C05453=1086.280,20.967,-58.503,174.648,18.923,153.065
C05454=1086.286,21.217,-58.517,174.650,18.926,153.065
C05455=1086.291,21.466,-58.532,174.652,18.928,153.065
C05456=1086.298,21.715,-58.547,174.653,18.929,153.065
C05457=1086.303,21.965,-58.562,174.654,18.931,153.065
C05458=1086.309,22.215,-58.576,174.656,18.933,153.065
C05459=1086.315,22.464,-58.591,174.658,18.935,153.065
C05460=1086.320,22.714,-58.606,174.659,18.937,153.065
C05461=1086.326,22.963,-58.621,174.661,18.939,153.065
C05462=1086.332,23.213,-58.635,174.663,18.941,153.066
C05463=1086.337,23.462,-58.650,174.664,18.942,153.066
C05464=1086.344,23.712,-58.665,174.666,18.944,153.066
C05465=1086.349,23.961,-58.680,174.667,18.946,153.066
C05466=1086.354,24.210,-58.695,174.669,18.948,153.066
C05467=1086.361,24.460,-58.710,174.671,18.951,153.066
C05468=1086.366,24.709,-58.724,174.672,18.952,153.066
C05469=1086.372,24.959,-58.739,174.674,18.954,153.066
C05470=1086.378,25.208,-58.754,174.676,18.956,153.066
C05471=1086.384,25.458,-58.769,174.677,18.958,153.066
C05472=1086.389,25.707,-58.784,174.680,18.960,153.066
C05473=1086.395,25.957,-58.799,174.681,18.962,153.066
C05474=1086.401,26.206,-58.813,174.682,18.963,153.067
C05475=1086.407,26.456,-58.829,174.684,18.966,153.067
C05476=1086.412,26.705,-58.843,174.686,18.967,153.067
C05477=1086.419,26.955,-58.858,174.687,18.969,153.067
C05478=1086.424,27.205,-58.873,174.689,18.971,153.067
C05479=1086.430,27.454,-58.888,174.691,18.973,153.067
C05480=1086.436,27.704,-58.903,174.692,18.975,153.067
C05481=1086.442,27.953,-58.918,174.694,18.977,153.067
C05482=1086.448,28.203,-58.933,174.695,18.979,153.067
C05483=1086.453,28.452,-58.948,174.697,18.980,153.067
C05484=1086.459,28.702,-58.963,174.699,18.983,153.067
C05485=1086.464,28.951,-58.978,174.700,18.984,153.067
C05486=1086.471,29.200,-58.993,174.702,18.986,153.068
C05487=1086.476,29.450,-59.008,174.704,18.988,153.068
C05488=1086.482,29.699,-59.023,174.705,18.990,153.068
C05489=1086.487,29.949,-59.038,174.706,18.992,153.068
C05490=1086.494,30.198,-59.053,174.709,18.994,153.068
C05491=1086.499,30.448,-59.069,174.710,18.996,153.068
C05492=1086.505,30.697,-59.084,174.711,18.997,153.068
C05493=1086.512,30.975,-59.101,174.713,19.000,153.068
C05494=1086.518,31.253,-59.117,174.716,19.002,153.068
C05495=1086.524,31.531,-59.134,174.717,19.004,153.068
C05496=1086.530,31.809,-59.152,174.719,19.006,153.068
C05497=1086.536,32.058,-59.167,174.720,19.008,153.069
C05498=1086.542,32.308,-59.182,174.723,19.010,153.069
C05499=1086.548,32.557,-59.197,174.724,19.012,153.069
C05500=1086.554,32.807,-59.212,174.725,19.014,153.069
C05501=1086.559,33.056,-59.227,174.728,19.016,153.069
C05502=1086.565,33.306,-59.242,174.729,19.017,153.069
C05503=1086.571,33.555,-59.257,174.731,19.020,153.069
C05504=1086.576,33.805,-59.272,174.732,19.021,153.069
C05505=1086.582,34.055,-59.288,174.734,19.023,153.069
C05506=1086.588,34.303,-59.303,174.736,19.025,153.069
C05507=1086.594,34.553,-59.319,174.737,19.027,153.069
C05508=1086.600,34.802,-59.333,174.739,19.029,153.069
C05509=1086.605,35.052,-59.349,174.741,19.031,153.069
C05510=1086.612,35.302,-59.364,174.742,19.033,153.070
C05511=1086.617,35.551,-59.380,174.745,19.035,153.070
C05512=1086.623,35.801,-59.395,174.746,19.037,153.070
C05513=1086.629,36.050,-59.410,174.747,19.038,153.070
C05514=1086.634,36.299,-59.425,174.750,19.040,153.070
C05515=1086.640,36.549,-59.440,174.751,19.042,153.070
C05516=1086.646,36.798,-59.456,174.752,19.044,153.070
C05517=1086.651,37.048,-59.472,174.754,19.046,153.070
C05518=1086.658,37.297,-59.487,174.756,19.047,153.070
C05519=1086.663,37.547,-59.502,174.758,19.050,153.070
C05520=1086.669,37.796,-59.518,174.759,19.051,153.070
C05521=1086.675,38.046,-59.533,174.761,19.053,153.070
C05522=1086.680,38.295,-59.548,174.763,19.056,153.070
C05523=1086.686,38.545,-59.564,174.764,19.057,153.070
C05524=1086.692,38.794,-59.580,174.766,19.059,153.071
C05525=1086.698,39.043,-59.595,174.768,19.061,153.071
C05526=1086.703,39.293,-59.610,174.769,19.063,153.071
C05527=1086.709,39.543,-59.627,174.772,19.065,153.071
C05528=1086.714,39.792,-59.642,174.773,19.067,153.071
C05529=1086.721,40.041,-59.657,174.774,19.068,153.071
C05530=1086.727,40.291,-59.673,174.776,19.070,153.071
C05531=1086.732,40.540,-59.688,174.778,19.072,153.071
C05532=1086.737,40.790,-59.704,174.780,19.074,153.071
C05533=1086.744,41.039,-59.719,174.781,19.076,153.071
C05534=1086.749,41.288,-59.734,174.783,19.078,153.071
C05535=1086.755,41.538,-59.750,174.785,19.080,153.071
C05536=1086.761,41.788,-59.766,174.786,19.081,153.071
C05537=1086.766,42.037,-59.781,174.788,19.084,153.072
C05538=1086.772,42.286,-59.797,174.790,19.086,153.072
C05539=1086.778,42.536,-59.813,174.791,19.087,153.072
C05540=1086.783,42.785,-59.828,174.793,19.090,153.072
C05541=1086.789,43.035,-59.844,174.795,19.091,153.072
C05542=1086.795,43.285,-59.860,174.796,19.093,153.072
C05543=1086.801,43.534,-59.876,174.798,19.095,153.072
C05544=1086.806,43.783,-59.890,174.800,19.097,153.072
C05545=1086.812,44.032,-59.907,174.802,19.099,153.072
C05546=1086.818,44.282,-59.922,174.803,19.100,153.072
C05547=1086.823,44.531,-59.938,174.805,19.102,153.072
C05548=1086.829,44.781,-59.954,174.807,19.104,153.072
C05549=1086.835,45.030,-59.970,174.808,19.106,153.072
C05550=1086.840,45.279,-59.985,174.810,19.108,153.073
C05551=1086.846,45.529,-60.001,174.812,19.110,153.073
C05552=1086.852,45.779,-60.017,174.814,19.112,153.073
C05553=1086.857,46.027,-60.033,174.815,19.114,153.073
C05554=1086.863,46.277,-60.048,174.817,19.116,153.073
C05555=1086.868,46.527,-60.065,174.819,19.118,153.073
C05556=1086.874,46.777,-60.080,174.820,19.120,153.073
C05557=1086.880,47.055,-60.098,174.822,19.122,153.073
C05558=1086.886,47.333,-60.116,174.825,19.124,153.073
C05559=1086.893,47.610,-60.133,174.826,19.126,153.073
C05560=1086.899,47.888,-60.151,174.828,19.128,153.073
C05561=1086.904,48.138,-60.167,174.829,19.130,153.073
C05562=1086.910,48.387,-60.183,174.832,19.132,153.073
C05563=1086.916,48.636,-60.199,174.833,19.134,153.074
C05564=1086.921,48.886,-60.214,174.835,19.136,153.074
C05565=1086.927,49.135,-60.231,174.837,19.137,153.074
C05566=1086.932,49.385,-60.246,174.838,19.139,153.074
C05567=1086.938,49.634,-60.262,174.840,19.141,153.074
C05568=1086.944,49.883,-60.278,174.842,19.143,153.074
C05569=1086.950,50.133,-60.294,174.844,19.145,153.074
C05570=1086.956,50.383,-60.310,174.845,19.147,153.074
C05571=1086.961,50.631,-60.326,174.847,19.149,153.074
C05572=1086.967,50.881,-60.342,174.849,19.151,153.074
C05573=1086.972,51.131,-60.358,174.850,19.152,153.074
C05574=1086.978,51.380,-60.375,174.853,19.154,153.074
C05575=1086.984,51.630,-60.390,174.854,19.156,153.074
C05576=1086.989,51.879,-60.406,174.856,19.158,153.074
C05577=1086.995,52.128,-60.422,174.857,19.160,153.074
C05578=1087.001,52.378,-60.439,174.860,19.162,153.074
C05579=1087.007,52.628,-60.454,174.861,19.164,153.075
C05580=1087.013,52.877,-60.470,174.862,19.165,153.075
C05581=1087.018,53.126,-60.486,174.865,19.167,153.075
C05582=1087.024,53.375,-60.503,174.866,19.169,153.075
C05583=1087.029,53.625,-60.518,174.868,19.171,153.075
C05584=1087.035,53.875,-60.535,174.870,19.173,153.075
C05585=1087.041,54.124,-60.551,174.872,19.175,153.075
C05586=1087.047,54.373,-60.568,174.873,19.176,153.075
C05587=1087.053,54.623,-60.584,174.875,19.178,153.075
C05588=1087.058,54.872,-60.599,174.877,19.180,153.075
C05589=1087.064,55.121,-60.615,174.878,19.182,153.075
C05590=1087.069,55.371,-60.631,174.881,19.184,153.075
C05591=1087.075,55.620,-60.648,174.882,19.186,153.075
C05592=1087.081,55.870,-60.665,174.884,19.188,153.075
C05593=1087.087,56.119,-60.681,174.886,19.189,153.075
C05594=1087.092,56.369,-60.696,174.887,19.191,153.075
C05595=1087.098,56.618,-60.713,174.890,19.193,153.075
C05596=1087.104,56.868,-60.729,174.891,19.195,153.076
C05597=1087.110,57.117,-60.745,174.893,19.197,153.076
C05598=1087.115,57.366,-60.761,174.894,19.198,153.076
C05599=1087.121,57.615,-60.778,174.897,19.200,153.076
C05600=1087.127,57.865,-60.794,174.898,19.202,153.076
C05601=1087.133,58.114,-60.810,174.901,19.204,153.076
C05602=1087.139,58.363,-60.827,174.902,19.205,153.076
C05603=1087.144,58.613,-60.843,174.903,19.207,153.076
C05604=1087.150,58.862,-60.859,174.905,19.209,153.076
C05605=1087.155,59.112,-60.875,174.907,19.211,153.076
C05606=1087.161,59.362,-60.892,174.909,19.213,153.076
C05607=1087.167,59.611,-60.908,174.911,19.215,153.076
C05608=1087.173,59.860,-60.924,174.913,19.217,153.076
C05609=1087.179,60.110,-60.940,174.914,19.218,153.076
C05610=1087.184,60.359,-60.957,174.917,19.220,153.076
C05611=1087.190,60.609,-60.973,174.918,19.222,153.076
C05612=1087.196,60.858,-60.990,174.920,19.224,153.076
C05613=1087.202,61.107,-61.006,174.922,19.225,153.076
C05614=1087.208,61.357,-61.022,174.923,19.227,153.076
C05615=1087.214,61.606,-61.040,174.926,19.229,153.076
C05616=1087.220,61.855,-61.056,174.927,19.230,153.076
C05617=1087.226,62.104,-61.072,174.929,19.233,153.076
C05618=1087.232,62.354,-61.089,174.931,19.234,153.076
C05619=1087.237,62.603,-61.105,174.933,19.236,153.076
C05620=1087.243,62.853,-61.122,174.934,19.238,153.076
C05621=1087.249,63.130,-61.140,174.937,19.240,153.076
C05622=1087.256,63.408,-61.158,174.939,19.242,153.076
C05623=1087.262,63.686,-61.176,174.940,19.243,153.077
C05624=1087.269,63.964,-61.195,174.943,19.245,153.077
C05625=1087.275,64.213,-61.211,174.945,19.247,153.077
C05626=1087.280,64.462,-61.228,174.946,19.249,153.077
C05627=1087.286,64.712,-61.245,174.948,19.251,153.077
C05628=1087.292,64.961,-61.261,174.950,19.253,153.077
C05629=1087.297,65.211,-61.278,174.952,19.254,153.077
C05630=1087.303,65.460,-61.294,174.954,19.256,153.077
C05631=1087.308,65.710,-61.311,174.955,19.258,153.077
C05632=1087.315,65.958,-61.328,174.957,19.260,153.077
C05633=1087.320,66.208,-61.345,174.959,19.262,153.077
C05634=1087.326,66.457,-61.361,174.961,19.264,153.077
C05635=1087.332,66.707,-61.377,174.963,19.265,153.077
C05636=1087.337,66.956,-61.394,174.965,19.267,153.077
C05637=1087.344,67.206,-61.411,174.966,19.269,153.077
C05638=1087.349,67.455,-61.428,174.969,19.271,153.077
C05639=1087.355,67.705,-61.444,174.970,19.272,153.077
C05640=1087.360,67.954,-61.461,174.972,19.274,153.077
C05641=1087.366,68.203,-61.478,174.974,19.276,153.077
C05642=1087.372,68.453,-61.495,174.976,19.278,153.077
C05643=1087.378,68.702,-61.511,174.978,19.279,153.077
C05644=1087.383,68.952,-61.528,174.980,19.281,153.077
C05645=1087.389,69.201,-61.545,174.981,19.283,153.077
C05646=1087.394,69.450,-61.562,174.984,19.285,153.077
C05647=1087.400,69.700,-61.578,174.985,19.286,153.077
C05648=1087.406,69.949,-61.596,174.987,19.288,153.077
C05649=1087.412,70.198,-61.612,174.989,19.290,153.077
C05650=1087.417,70.448,-61.629,174.990,19.292,153.077
C05651=1087.422,70.697,-61.647,174.992,19.294,153.077
C05652=1087.428,70.946,-61.663,174.994,19.295,153.077
C05653=1087.434,71.196,-61.680,174.996,19.297,153.077
C05654=1087.440,71.445,-61.697,174.998,19.299,153.078
C05655=1087.446,71.695,-61.714,175.000,19.301,153.078
C05656=1087.451,71.944,-61.731,175.001,19.302,153.078
C05657=1087.457,72.193,-61.748,175.004,19.304,153.078
C05658=1087.462,72.443,-61.765,175.005,19.306,153.078
C05659=1087.469,72.691,-61.782,175.007,19.308,153.078
C05660=1087.474,72.941,-61.798,175.009,19.309,153.078
C05661=1087.479,73.191,-61.815,175.011,19.311,153.078
C05662=1087.485,73.440,-61.832,175.013,19.313,153.078
C05663=1087.490,73.689,-61.849,175.015,19.315,153.078
C05664=1087.497,73.939,-61.867,175.016,19.316,153.078
C05665=1087.503,74.188,-61.883,175.019,19.318,153.078
C05666=1087.508,74.437,-61.901,175.020,19.320,153.078
C05667=1087.513,74.687,-61.918,175.022,19.322,153.078
C05668=1087.520,74.936,-61.935,175.024,19.323,153.078
C05669=1087.525,75.185,-61.951,175.026,19.325,153.078
C05670=1087.530,75.434,-61.969,175.028,19.327,153.078
C05671=1087.537,75.684,-61.986,175.030,19.329,153.078
C05672=1087.542,75.934,-62.003,175.031,19.330,153.078
C05673=1087.548,76.183,-62.020,175.034,19.332,153.078
C05674=1087.554,76.432,-62.037,175.035,19.334,153.078
C05675=1087.559,76.682,-62.054,175.038,19.336,153.078
C05676=1087.565,76.931,-62.071,175.039,19.337,153.078
C05677=1087.571,77.180,-62.089,175.041,19.339,153.078
C05678=1087.577,77.430,-62.106,175.043,19.341,153.078
C05679=1087.582,77.679,-62.123,175.045,19.343,153.078
C05680=1087.587,77.928,-62.140,175.047,19.344,153.078
C05681=1087.593,78.177,-62.158,175.049,19.346,153.078
C05682=1087.599,78.427,-62.174,175.051,19.348,153.078
C05683=1087.605,78.677,-62.192,175.053,19.350,153.078
C05684=1087.610,78.926,-62.209,175.055,19.352,153.078
C05685=1087.617,79.203,-62.228,175.056,19.353,153.078
C05686=1087.623,79.481,-62.248,175.059,19.355,153.078
C05687=1087.629,79.758,-62.266,175.061,19.357,153.078
C05688=1087.636,80.036,-62.287,175.063,19.359,153.078
C05689=1087.641,80.286,-62.303,175.065,19.361,153.078
C05690=1087.646,80.535,-62.321,175.067,19.363,153.078
C05691=1087.652,80.784,-62.339,175.069,19.364,153.078
C05692=1087.657,81.034,-62.355,175.071,19.366,153.078
C05693=1087.664,81.283,-62.373,175.073,19.367,153.078
C05694=1087.669,81.532,-62.390,175.075,19.369,153.078
C05695=1087.675,81.782,-62.407,175.076,19.371,153.078
C05696=1087.680,82.031,-62.425,175.079,19.373,153.078
C05697=1087.689,82.421,-62.453,175.082,19.375,153.078
C05698=1087.698,82.811,-62.480,175.085,19.378,153.078
C05699=1087.707,83.200,-62.506,175.088,19.381,153.078
C05700=1087.716,83.590,-62.534,175.091,19.384,153.078
C05701=1087.721,83.839,-62.551,175.092,19.385,153.078
C05702=1087.727,84.089,-62.569,175.095,19.387,153.078
C05703=1087.733,84.338,-62.587,175.096,19.389,153.078
C05704=1087.738,84.587,-62.604,175.098,19.391,153.078
C05705=1087.744,84.836,-62.622,175.100,19.392,153.078
C05706=1087.750,85.086,-62.640,175.102,19.394,153.078
C05707=1087.755,85.336,-62.656,175.105,19.396,153.078
C05708=1087.761,85.585,-62.674,175.106,19.397,153.078
C05709=1087.767,85.835,-62.692,175.108,19.399,153.078
C05710=1087.772,86.084,-62.710,175.110,19.401,153.078
C05711=1087.778,86.333,-62.727,175.112,19.402,153.078
C05712=1087.783,86.582,-62.745,175.114,19.404,153.078
C05713=1087.789,86.831,-62.763,175.116,19.406,153.078
C05714=1087.795,87.080,-62.780,175.118,19.407,153.078
C05715=1087.800,87.329,-62.798,175.120,19.409,153.078
C05716=1087.806,87.580,-62.815,175.122,19.410,153.078
C05717=1087.812,87.829,-62.832,175.124,19.412,153.078
C05718=1087.817,88.078,-62.850,175.126,19.414,153.078
C05719=1087.823,88.328,-62.868,175.128,19.415,153.078
C05720=1087.829,88.577,-62.886,175.130,19.417,153.078
C05721=1087.834,88.826,-62.903,175.132,19.419,153.078
C05722=1087.840,89.075,-62.921,175.134,19.421,153.078
C05723=1087.846,89.325,-62.939,175.136,19.422,153.078
C05724=1087.852,89.574,-62.957,175.138,19.424,153.078
C05725=1087.858,89.823,-62.974,175.139,19.425,153.078
C05726=1087.863,90.072,-62.992,175.142,19.427,153.078
C05727=1087.869,90.322,-63.010,175.144,19.429,153.078
C05728=1087.875,90.571,-63.027,175.146,19.430,153.078
C05729=1087.880,90.820,-63.045,175.148,19.432,153.078
C05730=1087.886,91.070,-63.063,175.150,19.434,153.078
C05731=1087.892,91.319,-63.080,175.152,19.436,153.078
C05732=1087.897,91.568,-63.098,175.153,19.437,153.078
C05733=1087.903,91.817,-63.117,175.156,19.439,153.078
C05734=1087.909,92.066,-63.135,175.157,19.440,153.078
C05735=1087.915,92.316,-63.153,175.160,19.442,153.078
C05736=1087.920,92.565,-63.170,175.162,19.444,153.078
C05737=1087.925,92.815,-63.188,175.164,19.445,153.078
C05738=1087.931,93.064,-63.206,175.166,19.447,153.078
C05739=1087.937,93.313,-63.224,175.168,19.449,153.078
C05740=1087.942,93.562,-63.241,175.170,19.451,153.078
C05741=1087.948,93.812,-63.259,175.172,19.452,153.078
C05742=1087.953,94.061,-63.278,175.174,19.454,153.078
C05743=1087.959,94.310,-63.296,175.176,19.456,153.078
C05744=1087.965,94.560,-63.314,175.178,19.457,153.078
C05745=1087.974,94.947,-63.342,175.181,19.459,153.078
C05746=1087.982,95.333,-63.370,175.184,19.462,153.078
C05747=1087.991,95.720,-63.398,175.187,19.465,153.078
C05748=1088.000,96.106,-63.425,175.190,19.467,153.078
C05749=1088.006,96.355,-63.444,175.193,19.469,153.078
C05750=1088.011,96.604,-63.462,175.194,19.470,153.078
C05751=1088.017,96.854,-63.480,175.197,19.472,153.078
C05752=1088.022,97.103,-63.497,175.198,19.473,153.078
C05753=1088.028,97.353,-63.517,175.200,19.475,153.078
C05754=1088.034,97.602,-63.534,175.203,19.477,153.078
C05755=1088.040,97.851,-63.552,175.204,19.478,153.078
C05756=1088.046,98.100,-63.570,175.207,19.480,153.078
C05757=1088.051,98.350,-63.589,175.208,19.481,153.078
C05758=1088.056,98.599,-63.606,175.211,19.483,153.078
C05759=1088.063,98.849,-63.624,175.213,19.485,153.078
C05760=1088.068,99.097,-63.643,175.215,19.486,153.078
C05761=1088.073,99.346,-63.661,175.217,19.488,153.077
C05762=1088.079,99.596,-63.679,175.219,19.490,153.078
C05763=1088.085,99.846,-63.698,175.221,19.492,153.078
C05764=1088.090,100.095,-63.716,175.224,19.493,153.077
C05765=1088.097,100.344,-63.734,175.225,19.495,153.077
C05766=1088.102,100.593,-63.752,175.228,19.496,153.077
C05767=1088.108,100.843,-63.770,175.229,19.498,153.077
C05768=1088.114,101.091,-63.789,175.232,19.499,153.077
C05769=1088.119,101.341,-63.807,175.234,19.501,153.077
C05770=1088.125,101.590,-63.825,175.236,19.502,153.077
C05771=1088.130,101.840,-63.844,175.238,19.504,153.077
C05772=1088.136,102.088,-63.862,175.239,19.506,153.077
C05773=1088.141,102.338,-63.881,175.242,19.507,153.077
C05774=1088.147,102.587,-63.898,175.244,19.509,153.077
C05775=1088.153,102.837,-63.918,175.246,19.510,153.077
C05776=1088.158,103.086,-63.935,175.248,19.512,153.077
C05777=1088.164,103.335,-63.954,175.250,19.513,153.077
C05778=1088.169,103.584,-63.972,175.252,19.515,153.077
C05779=1088.175,103.834,-63.991,175.255,19.517,153.077
C05780=1088.181,104.083,-64.009,175.256,19.518,153.077
C05781=1088.186,104.332,-64.028,175.259,19.520,153.077
C05782=1088.192,104.581,-64.046,175.260,19.521,153.077
C05783=1088.197,104.831,-64.065,175.263,19.523,153.077
C05784=1088.203,105.079,-64.083,175.265,19.525,153.077
C05785=1088.209,105.329,-64.102,175.267,19.526,153.077
C05786=1088.214,105.578,-64.120,175.269,19.528,153.077
C05787=1088.220,105.828,-64.138,175.271,19.530,153.077
C05788=1088.226,106.077,-64.158,175.273,19.531,153.077
C05789=1088.231,106.326,-64.175,175.275,19.533,153.077
C05790=1088.237,106.575,-64.194,175.277,19.534,153.076
C05791=1088.243,106.824,-64.213,175.279,19.536,153.076
C05792=1088.248,107.074,-64.231,175.282,19.537,153.076
C05793=1088.253,107.323,-64.250,175.283,19.539,153.076
C05794=1088.259,107.572,-64.269,175.286,19.540,153.076
C05795=1088.265,107.822,-64.287,175.287,19.542,153.076
C05796=1088.271,108.070,-64.306,175.290,19.543,153.076
C05797=1088.276,108.320,-64.324,175.292,19.545,153.076
C05798=1088.282,108.570,-64.343,175.294,19.546,153.076
C05799=1088.288,108.818,-64.362,175.296,19.548,153.076
C05800=1088.293,109.068,-64.381,175.299,19.550,153.076
C05801=1088.299,109.317,-64.398,175.300,19.551,153.076
C05802=1088.304,109.566,-64.418,175.303,19.553,153.076
C05803=1088.310,109.816,-64.437,175.305,19.555,153.076
C05804=1088.316,110.065,-64.455,175.307,19.556,153.076
C05805=1088.321,110.314,-64.474,175.309,19.558,153.076
C05806=1088.328,110.563,-64.492,175.311,19.559,153.076
C05807=1088.333,110.812,-64.511,175.314,19.560,153.075
C05808=1088.338,111.062,-64.530,175.316,19.562,153.075
C05809=1088.345,111.339,-64.551,175.318,19.564,153.075
C05810=1088.351,111.617,-64.572,175.321,19.566,153.075
C05811=1088.358,111.895,-64.593,175.323,19.567,153.075
C05812=1088.364,112.173,-64.614,175.325,19.568,153.075
C05813=1088.369,112.422,-64.633,175.327,19.570,153.075
C05814=1088.375,112.671,-64.652,175.330,19.572,153.075
C05815=1088.381,112.921,-64.670,175.331,19.573,153.075
C05816=1088.386,113.170,-64.689,175.334,19.575,153.075
C05817=1088.392,113.419,-64.708,175.336,19.576,153.075
C05818=1088.398,113.668,-64.727,175.338,19.578,153.075
C05819=1088.403,113.917,-64.746,175.340,19.579,153.075
C05820=1088.409,114.166,-64.765,175.343,19.581,153.075
C05821=1088.414,114.416,-64.784,175.344,19.582,153.075
C05822=1088.420,114.664,-64.803,175.347,19.584,153.075
C05823=1088.426,114.914,-64.821,175.349,19.586,153.075
C05824=1088.431,115.164,-64.840,175.351,19.587,153.074
C05825=1088.436,115.412,-64.859,175.353,19.588,153.074
C05826=1088.442,115.662,-64.878,175.356,19.590,153.074
C05827=1088.448,115.911,-64.898,175.357,19.591,153.074
C05828=1088.453,116.160,-64.917,175.360,19.593,153.074
C05829=1088.459,116.409,-64.936,175.362,19.595,153.074
C05830=1088.464,116.659,-64.955,175.364,19.596,153.074
C05831=1088.469,116.908,-64.974,175.366,19.598,153.074
C05832=1088.475,117.157,-64.993,175.369,19.599,153.074
C05833=1088.481,117.406,-65.012,175.371,19.600,153.074
C05834=1088.486,117.656,-65.032,175.373,19.602,153.074
C05835=1088.491,117.905,-65.051,175.375,19.604,153.074
C05836=1088.497,118.154,-65.070,175.377,19.605,153.074
C05837=1088.503,118.403,-65.089,175.379,19.607,153.074
C05838=1088.508,118.652,-65.108,175.382,19.608,153.074
C05839=1088.514,118.902,-65.127,175.384,19.609,153.073
C05840=1088.519,119.151,-65.146,175.386,19.611,153.073
C05841=1088.525,119.400,-65.166,175.388,19.613,153.073
C05842=1088.530,119.649,-65.185,175.390,19.614,153.073
C05843=1088.536,119.898,-65.204,175.392,19.616,153.073
C05844=1088.542,120.147,-65.224,175.395,19.617,153.073
C05845=1088.547,120.397,-65.243,175.397,19.618,153.073
C05846=1088.553,120.646,-65.262,175.399,19.620,153.073
C05847=1088.558,120.895,-65.281,175.402,19.622,153.073
C05848=1088.564,121.144,-65.300,175.403,19.623,153.073
C05849=1088.570,121.394,-65.320,175.406,19.625,153.073
C05850=1088.575,121.643,-65.339,175.408,19.627,153.073
C05851=1088.581,121.891,-65.358,175.410,19.628,153.073
C05852=1088.586,122.141,-65.378,175.412,19.629,153.073
C05853=1088.592,122.390,-65.397,175.415,19.631,153.072
C05854=1088.598,122.640,-65.416,175.417,19.632,153.072
C05855=1088.603,122.889,-65.435,175.419,19.634,153.072
C05856=1088.609,123.137,-65.455,175.421,19.635,153.072
C05857=1088.615,123.387,-65.474,175.424,19.637,153.072
C05858=1088.620,123.636,-65.493,175.426,19.638,153.072
C05859=1088.626,123.886,-65.513,175.428,19.639,153.072
C05860=1088.632,124.134,-65.533,175.431,19.641,153.072
C05861=1088.638,124.384,-65.552,175.432,19.642,153.072
C05862=1088.643,124.633,-65.571,175.435,19.644,153.072
C05863=1088.648,124.882,-65.590,175.437,19.645,153.072
C05864=1088.654,125.131,-65.611,175.439,19.646,153.071
C05865=1088.659,125.381,-65.630,175.442,19.648,153.071
C05866=1088.665,125.630,-65.649,175.444,19.649,153.071
C05867=1088.671,125.879,-65.669,175.446,19.651,153.071
C05868=1088.677,126.128,-65.688,175.448,19.652,153.071
C05869=1088.682,126.378,-65.708,175.451,19.654,153.071
C05870=1088.688,126.626,-65.727,175.453,19.655,153.071
C05871=1088.693,126.875,-65.746,175.455,19.656,153.071
C05872=1088.699,127.125,-65.766,175.457,19.658,153.071
C05873=1088.706,127.402,-65.788,175.460,19.659,153.071
C05874=1088.712,127.680,-65.810,175.463,19.661,153.070
C05875=1088.718,127.958,-65.831,175.465,19.662,153.070
C05876=1088.725,128.235,-65.854,175.468,19.664,153.070
C05877=1088.730,128.485,-65.873,175.470,19.666,153.070
C05878=1088.735,128.734,-65.893,175.473,19.667,153.070
C05879=1088.741,128.983,-65.913,175.474,19.668,153.070
C05880=1088.747,129.233,-65.932,175.477,19.670,153.070
C05881=1088.753,129.481,-65.952,175.479,19.671,153.070
C05882=1088.759,129.731,-65.971,175.481,19.672,153.070
C05883=1088.765,129.980,-65.991,175.484,19.674,153.069
C05884=1088.770,130.229,-66.010,175.486,19.675,153.069
C05885=1088.776,130.478,-66.031,175.489,19.677,153.069
C05886=1088.781,130.728,-66.050,175.490,19.678,153.069
C05887=1088.787,130.976,-66.070,175.493,19.679,153.069
C05888=1088.793,131.226,-66.089,175.495,19.681,153.069
C05889=1088.799,131.475,-66.109,175.498,19.682,153.069
C05890=1088.804,131.724,-66.129,175.500,19.683,153.069
C05891=1088.810,131.973,-66.149,175.502,19.685,153.069
C05892=1088.816,132.222,-66.169,175.505,19.686,153.068
C05893=1088.822,132.471,-66.188,175.506,19.687,153.068
C05894=1088.827,132.721,-66.209,175.509,19.689,153.068
C05895=1088.833,132.970,-66.228,175.512,19.691,153.068
C05896=1088.839,133.219,-66.248,175.514,19.692,153.068
C05897=1088.844,133.468,-66.268,175.516,19.693,153.068
C05898=1088.850,133.717,-66.288,175.518,19.695,153.068
C05899=1088.855,133.967,-66.308,175.521,19.696,153.068
C05900=1088.860,134.215,-66.327,175.523,19.698,153.067
C05901=1088.866,134.464,-66.347,175.525,19.699,153.067
C05902=1088.871,134.713,-66.368,175.528,19.700,153.067
C05903=1088.877,134.963,-66.387,175.530,19.702,153.067
C05904=1088.882,135.212,-66.407,175.533,19.703,153.067
C05905=1088.888,135.461,-66.427,175.534,19.704,153.067
C05906=1088.894,135.710,-66.447,175.537,19.706,153.067
C05907=1088.900,135.960,-66.468,175.540,19.707,153.067
C05908=1088.906,136.209,-66.488,175.542,19.709,153.067
C05909=1088.911,136.458,-66.508,175.544,19.710,153.066
C05910=1088.917,136.707,-66.527,175.546,19.711,153.066
C05911=1088.923,136.956,-66.547,175.549,19.713,153.066
C05912=1088.928,137.205,-66.568,175.551,19.714,153.066
C05913=1088.934,137.454,-66.588,175.553,19.715,153.066
C05914=1088.939,137.704,-66.608,175.556,19.716,153.066
C05915=1088.945,137.953,-66.628,175.558,19.718,153.066
C05916=1088.950,138.202,-66.648,175.561,19.719,153.066
C05917=1088.956,138.450,-66.668,175.563,19.720,153.065
C05918=1088.961,138.700,-66.689,175.565,19.722,153.065
C05919=1088.967,138.949,-66.708,175.568,19.723,153.065
C05920=1088.972,139.198,-66.728,175.570,19.725,153.065
C05921=1088.978,139.447,-66.748,175.572,19.726,153.065
C05922=1088.983,139.696,-66.769,175.575,19.727,153.065
C05923=1088.989,139.945,-66.789,175.577,19.729,153.065
C05924=1088.995,140.195,-66.810,175.580,19.730,153.065
C05925=1089.001,140.444,-66.830,175.582,19.731,153.064
C05926=1089.007,140.693,-66.850,175.584,19.732,153.064
C05927=1089.012,140.942,-66.870,175.587,19.734,153.064
C05928=1089.018,141.191,-66.890,175.589,19.735,153.064
C05929=1089.023,141.440,-66.911,175.592,19.737,153.064
C05930=1089.029,141.689,-66.931,175.594,19.738,153.064
C05931=1089.034,141.938,-66.951,175.596,19.739,153.064
C05932=1089.039,142.187,-66.972,175.599,19.741,153.064
C05933=1089.045,142.436,-66.992,175.601,19.742,153.063
C05934=1089.051,142.685,-67.012,175.604,19.744,153.063
C05935=1089.056,142.935,-67.033,175.606,19.744,153.063
C05936=1089.062,143.184,-67.053,175.608,19.746,153.063
C05937=1089.068,143.461,-67.076,175.611,19.747,153.063
C05938=1089.075,143.739,-67.098,175.613,19.749,153.063
C05939=1089.081,144.017,-67.122,175.616,19.750,153.063
C05940=1089.086,144.294,-67.144,175.619,19.753,153.062
C05941=1089.093,144.544,-67.165,175.621,19.753,153.062
C05942=1089.098,144.793,-67.185,175.624,19.755,153.062
C05943=1089.104,145.042,-67.206,175.626,19.756,153.062
C05944=1089.109,145.291,-67.226,175.629,19.758,153.062
C05945=1089.115,145.540,-67.246,175.631,19.759,153.062
C05946=1089.120,145.789,-67.267,175.633,19.760,153.061
C05947=1089.126,146.039,-67.288,175.636,19.761,153.061
C05948=1089.132,146.287,-67.308,175.638,19.763,153.061
C05949=1089.137,146.536,-67.329,175.641,19.764,153.061
C05950=1089.143,146.785,-67.350,175.643,19.766,153.061
C05951=1089.149,147.034,-67.370,175.645,19.766,153.061
C05952=1089.155,147.284,-67.390,175.648,19.768,153.061
C05953=1089.160,147.533,-67.411,175.650,19.769,153.061
C05954=1089.165,147.781,-67.432,175.653,19.770,153.060
C05955=1089.171,148.030,-67.452,175.656,19.772,153.060
C05956=1089.177,148.280,-67.473,175.658,19.773,153.060
C05957=1089.182,148.529,-67.494,175.660,19.774,153.060
C05958=1089.188,148.778,-67.514,175.663,19.776,153.060
C05959=1089.194,149.027,-67.535,175.665,19.777,153.060
C05960=1089.199,149.276,-67.555,175.668,19.778,153.059
C05961=1089.205,149.526,-67.576,175.670,19.779,153.059
C05962=1089.210,149.775,-67.597,175.672,19.781,153.059
C05963=1089.216,150.023,-67.618,175.675,19.782,153.059
C05964=1089.221,150.272,-67.639,175.678,19.783,153.059
C05965=1089.227,150.522,-67.660,175.680,19.785,153.059
C05966=1089.232,150.771,-67.680,175.683,19.786,153.058
C05967=1089.239,151.019,-67.701,175.685,19.787,153.058
C05968=1089.244,151.269,-67.721,175.687,19.788,153.058
C05969=1089.249,151.518,-67.742,175.690,19.790,153.058
C05970=1089.255,151.767,-67.764,175.692,19.791,153.058
C05971=1089.261,152.016,-67.784,175.695,19.792,153.058
C05972=1089.266,152.265,-67.805,175.698,19.794,153.058
C05973=1089.272,152.514,-67.826,175.699,19.795,153.058
C05974=1089.277,152.763,-67.847,175.702,19.796,153.057
C05975=1089.283,153.012,-67.868,175.705,19.797,153.057
C05976=1089.288,153.261,-67.889,175.707,19.799,153.057
C05977=1089.294,153.511,-67.910,175.710,19.800,153.057
C05978=1089.299,153.759,-67.931,175.712,19.801,153.057
C05979=1089.305,154.009,-67.952,175.714,19.803,153.057
C05980=1089.311,154.258,-67.973,175.717,19.804,153.056
C05981=1089.316,154.507,-67.994,175.719,19.805,153.056
C05982=1089.322,154.755,-68.015,175.722,19.807,153.056
C05983=1089.328,155.005,-68.035,175.725,19.808,153.056
C05984=1089.334,155.254,-68.056,175.727,19.809,153.056
C05985=1089.339,155.502,-68.077,175.729,19.810,153.055
C05986=1089.345,155.752,-68.098,175.732,19.811,153.055
C05987=1089.350,156.001,-68.120,175.734,19.813,153.055
C05988=1089.355,156.250,-68.140,175.737,19.814,153.055
C05989=1089.361,156.499,-68.162,175.740,19.815,153.055
C05990=1089.367,156.748,-68.183,175.742,19.817,153.055
C05991=1089.372,156.997,-68.204,175.745,19.818,153.054
C05992=1089.378,157.246,-68.225,175.747,19.819,153.054
C05993=1089.383,157.495,-68.246,175.749,19.820,153.054
C05994=1089.389,157.744,-68.267,175.752,19.821,153.054
C05995=1089.395,157.994,-68.288,175.755,19.823,153.054
C05996=1089.400,158.242,-68.310,175.757,19.824,153.054
C05997=1089.406,158.491,-68.331,175.760,19.825,153.053
C05998=1089.412,158.741,-68.352,175.762,19.827,153.053
C05999=1089.417,158.989,-68.374,175.765,19.828,153.053
C06000=1089.422,159.239,-68.394,175.767,19.829,153.053
C06001=1089.428,159.516,-68.418,175.771,19.830,153.053
C06002=1089.435,159.793,-68.442,175.773,19.832,153.053
C06003=1089.441,160.071,-68.466,175.776,19.833,153.052
C06004=1089.448,160.348,-68.490,175.778,19.834,153.052
C06005=1089.453,160.597,-68.510,175.781,19.835,153.052
C06006=1089.459,160.846,-68.532,175.784,19.837,153.052
C06007=1089.465,161.095,-68.553,175.787,19.838,153.052
C06008=1089.470,161.344,-68.575,175.789,19.839,153.051
C06009=1089.475,161.593,-68.596,175.792,19.840,153.051
C06010=1089.481,161.842,-68.617,175.794,19.841,153.051
C06011=1089.487,162.091,-68.639,175.796,19.843,153.051
C06012=1089.492,162.341,-68.660,175.799,19.844,153.051
C06013=1089.497,162.589,-68.681,175.801,19.846,153.051
C06014=1089.503,162.839,-68.703,175.804,19.847,153.050
C06015=1089.508,163.087,-68.725,175.807,19.848,153.050
C06016=1089.514,163.336,-68.746,175.809,19.850,153.050
C06017=1089.519,163.586,-68.767,175.812,19.851,153.050
C06018=1089.524,163.834,-68.789,175.815,19.852,153.050
C06019=1089.530,164.084,-68.811,175.817,19.854,153.050
C06020=1089.535,164.332,-68.832,175.819,19.854,153.049
C06021=1089.541,164.581,-68.854,175.822,19.856,153.049
C06022=1089.546,164.830,-68.876,175.824,19.857,153.049
C06023=1089.552,165.079,-68.897,175.827,19.858,153.049
C06024=1089.557,165.329,-68.918,175.830,19.860,153.049
C06025=1089.563,165.577,-68.940,175.832,19.861,153.049
C06026=1089.568,165.827,-68.962,175.835,19.862,153.048
C06027=1089.574,166.075,-68.983,175.837,19.864,153.048
C06028=1089.579,166.325,-69.005,175.840,19.865,153.048
C06029=1089.585,166.573,-69.027,175.843,19.866,153.048
C06030=1089.590,166.822,-69.048,175.846,19.867,153.048
C06031=1089.595,167.071,-69.070,175.847,19.868,153.048
C06032=1089.601,167.320,-69.091,175.850,19.869,153.047
C06033=1089.606,167.570,-69.114,175.853,19.871,153.047
C06034=1089.612,167.818,-69.135,175.855,19.872,153.047
C06035=1089.617,168.068,-69.157,175.858,19.873,153.047
C06036=1089.623,168.316,-69.178,175.861,19.874,153.047
C06037=1089.628,168.566,-69.201,175.863,19.876,153.046
C06038=1089.634,168.814,-69.222,175.866,19.877,153.046
C06039=1089.639,169.064,-69.244,175.869,19.878,153.046
C06040=1089.645,169.312,-69.265,175.871,19.879,153.046
C06041=1089.650,169.562,-69.288,175.874,19.881,153.046
C06042=1089.656,169.810,-69.309,175.877,19.882,153.045
C06043=1089.661,170.060,-69.331,175.879,19.884,153.045
C06044=1089.667,170.308,-69.352,175.882,19.885,153.045
C06045=1089.672,170.558,-69.375,175.884,19.886,153.045
C06046=1089.678,170.806,-69.397,175.887,19.887,153.045
C06047=1089.684,171.055,-69.419,175.889,19.888,153.044
C06048=1089.690,171.304,-69.441,175.892,19.889,153.044
C06049=1089.695,171.553,-69.462,175.895,19.890,153.044
C06050=1089.700,171.803,-69.485,175.897,19.892,153.044
C06051=1089.706,172.051,-69.506,175.900,19.893,153.044
C06052=1089.711,172.300,-69.529,175.903,19.894,153.044
C06053=1089.717,172.548,-69.550,175.905,19.895,153.043
C06054=1089.722,172.798,-69.572,175.908,19.896,153.043
C06055=1089.729,173.047,-69.594,175.911,19.898,153.043
C06056=1089.733,173.296,-69.616,175.913,19.899,153.043
C06057=1089.739,173.545,-69.639,175.916,19.900,153.043
C06058=1089.745,173.794,-69.660,175.919,19.901,153.042
C06059=1089.750,174.043,-69.682,175.922,19.902,153.042
C06060=1089.756,174.292,-69.704,175.924,19.904,153.042
C06061=1089.761,174.540,-69.727,175.927,19.905,153.042
C06062=1089.768,174.790,-69.748,175.930,19.906,153.041
C06063=1089.773,175.039,-69.770,175.932,19.907,153.041
C06064=1089.778,175.287,-69.793,175.935,19.908,153.041
C06065=1089.785,175.565,-69.817,175.938,19.909,153.041
C06066=1089.791,175.842,-69.842,175.941,19.910,153.041
C06067=1089.797,176.118,-69.867,175.943,19.912,153.040
C06068=1089.803,176.396,-69.891,175.947,19.914,153.040
C06069=1089.809,176.645,-69.913,175.949,19.915,153.040
C06070=1089.815,176.894,-69.936,175.952,19.916,153.040
C06071=1089.820,177.143,-69.957,175.955,19.917,153.040
C06072=1089.826,177.392,-69.980,175.958,19.918,153.039
C06073=1089.832,177.641,-70.002,175.960,19.919,153.039
C06074=1089.837,177.889,-70.025,175.963,19.921,153.039
C06075=1089.843,178.138,-70.046,175.966,19.922,153.039
C06076=1089.849,178.387,-70.069,175.968,19.923,153.038
C06077=1089.854,178.637,-70.091,175.971,19.924,153.038
C06078=1089.860,178.885,-70.113,175.974,19.925,153.038
C06079=1089.865,179.134,-70.136,175.976,19.926,153.038
C06080=1089.871,179.384,-70.158,175.979,19.927,153.038
C06081=1089.877,179.632,-70.180,175.981,19.928,153.037
C06082=1089.882,179.881,-70.203,175.984,19.929,153.037
C06083=1089.888,180.130,-70.225,175.987,19.930,153.037
C06084=1089.894,180.379,-70.247,175.989,19.931,153.037
C06085=1089.900,180.628,-70.270,175.992,19.932,153.036
C06086=1089.905,180.877,-70.293,175.995,19.933,153.036
C06087=1089.911,181.126,-70.314,175.998,19.934,153.036
C06088=1089.917,181.374,-70.337,176.000,19.936,153.036
C06089=1089.922,181.624,-70.359,176.003,19.937,153.036
C06090=1089.928,181.873,-70.382,176.006,19.938,153.035
C06091=1089.934,182.121,-70.404,176.009,19.939,153.035
C06092=1089.939,182.370,-70.426,176.011,19.940,153.035
C06093=1089.945,182.619,-70.449,176.014,19.941,153.034
C06094=1089.951,182.868,-70.471,176.017,19.943,153.034
C06095=1089.957,183.117,-70.494,176.020,19.944,153.034
C06096=1089.962,183.366,-70.517,176.022,19.945,153.034
C06097=1089.968,183.615,-70.540,176.025,19.946,153.034
C06098=1089.974,183.864,-70.561,176.028,19.947,153.033
C06099=1089.979,184.112,-70.584,176.031,19.948,153.033
C06100=1089.985,184.361,-70.607,176.034,19.949,153.033
C06101=1089.991,184.611,-70.629,176.037,19.950,153.033
C06102=1089.996,184.860,-70.652,176.040,19.951,153.032
C06103=1090.003,185.108,-70.674,176.042,19.953,153.032
C06104=1090.009,185.357,-70.697,176.045,19.954,153.032
C06105=1090.013,185.606,-70.720,176.048,19.955,153.032
C06106=1090.018,185.855,-70.743,176.050,19.956,153.032
C06107=1090.024,186.104,-70.766,176.053,19.957,153.031
C06108=1090.030,186.353,-70.788,176.056,19.958,153.031
C06109=1090.035,186.602,-70.810,176.059,19.960,153.031
C06110=1090.040,186.851,-70.833,176.061,19.961,153.031
C06111=1090.046,187.100,-70.856,176.064,19.962,153.030
C06112=1090.052,187.349,-70.879,176.067,19.963,153.030
C06113=1090.058,187.597,-70.902,176.069,19.965,153.030
C06114=1090.063,187.846,-70.925,176.072,19.966,153.030
C06115=1090.067,188.096,-70.948,176.075,19.967,153.030
C06116=1090.073,188.344,-70.970,176.078,19.968,153.029
C06117=1090.079,188.593,-70.993,176.080,19.969,153.029
C06118=1090.085,188.842,-71.016,176.083,19.970,153.029
C06119=1090.090,189.091,-71.039,176.086,19.971,153.029
C06120=1090.095,189.339,-71.062,176.089,19.972,153.028
C06121=1090.101,189.588,-71.085,176.091,19.974,153.028
C06122=1090.106,189.837,-71.108,176.094,19.975,153.028
C06123=1090.112,190.086,-71.131,176.097,19.976,153.028
C06124=1090.118,190.335,-71.154,176.100,19.977,153.028
C06125=1090.123,190.584,-71.177,176.103,19.978,153.027
C06126=1090.129,190.833,-71.200,176.106,19.980,153.027
C06127=1090.134,191.081,-71.223,176.109,19.981,153.027
C06128=1090.139,191.330,-71.246,176.111,19.982,153.027
C06129=1090.145,191.607,-71.271,176.114,19.983,153.026
C06130=1090.152,191.884,-71.297,176.118,19.985,153.026
C06131=1090.158,192.161,-71.322,176.121,19.986,153.026
C06132=1090.164,192.438,-71.349,176.123,19.987,153.026
C06133=1090.170,192.686,-71.371,176.127,19.988,153.025
C06134=1090.175,192.935,-71.394,176.129,19.990,153.025
C06135=1090.180,193.184,-71.418,176.132,19.991,153.025
C06136=1090.186,193.433,-71.441,176.135,19.992,153.025
C06137=1090.192,193.682,-71.464,176.138,19.993,153.024
C06138=1090.198,193.930,-71.487,176.141,19.994,153.024
C06139=1090.203,194.180,-71.511,176.143,19.995,153.024
C06140=1090.209,194.428,-71.534,176.146,19.996,153.024
C06141=1090.214,194.677,-71.557,176.149,19.997,153.024
C06142=1090.220,194.926,-71.580,176.152,19.998,153.023
C06143=1090.225,195.175,-71.603,176.154,19.999,153.023
C06144=1090.231,195.424,-71.627,176.157,20.001,153.023
C06145=1090.237,195.673,-71.650,176.161,20.002,153.023
C06146=1090.242,195.922,-71.673,176.163,20.003,153.022
C06147=1090.247,196.171,-71.696,176.166,20.004,153.022
C06148=1090.253,196.420,-71.719,176.169,20.005,153.022
C06149=1090.259,196.668,-71.743,176.172,20.006,153.022
C06150=1090.265,196.917,-71.766,176.175,20.007,153.021
C06151=1090.270,197.166,-71.789,176.177,20.008,153.021
C06152=1090.276,197.415,-71.812,176.180,20.009,153.021
C06153=1090.282,197.663,-71.836,176.183,20.011,153.021
C06154=1090.287,197.912,-71.860,176.186,20.012,153.020
C06155=1090.292,198.161,-71.882,176.189,20.013,153.020
C06156=1090.298,198.410,-71.906,176.192,20.014,153.020
C06157=1090.304,198.659,-71.930,176.195,20.015,153.020
C06158=1090.310,198.908,-71.953,176.197,20.016,153.019
C06159=1090.316,199.157,-71.977,176.200,20.017,153.019
C06160=1090.321,199.406,-72.000,176.203,20.019,153.019
C06161=1090.327,199.654,-72.024,176.206,20.020,153.019
C06162=1090.333,199.903,-72.047,176.209,20.021,153.018
C06163=1090.338,200.152,-72.070,176.212,20.022,153.018
C06164=1090.344,200.401,-72.094,176.215,20.023,153.018
C06165=1090.349,200.649,-72.117,176.218,20.024,153.018
C06166=1090.355,200.898,-72.141,176.221,20.025,153.017
C06167=1090.361,201.148,-72.165,176.223,20.026,153.017
C06168=1090.367,201.396,-72.188,176.226,20.027,153.017
C06169=1090.372,201.645,-72.212,176.229,20.028,153.017
C06170=1090.378,201.893,-72.235,176.232,20.029,153.016
C06171=1090.383,202.143,-72.259,176.235,20.031,153.016
C06172=1090.389,202.391,-72.283,176.238,20.032,153.016
C06173=1090.395,202.640,-72.306,176.241,20.033,153.016
C06174=1090.401,202.889,-72.330,176.244,20.034,153.015
C06175=1090.406,203.138,-72.353,176.246,20.035,153.015
C06176=1090.412,203.387,-72.377,176.249,20.036,153.015
C06177=1090.417,203.636,-72.401,176.253,20.038,153.015
C06178=1090.423,203.884,-72.425,176.256,20.039,153.014
C06179=1090.428,204.133,-72.448,176.258,20.040,153.014
C06180=1090.434,204.381,-72.472,176.261,20.041,153.014
C06181=1090.440,204.631,-72.496,176.264,20.042,153.014
C06182=1090.445,204.880,-72.520,176.267,20.043,153.013
C06183=1090.451,205.128,-72.544,176.269,20.044,153.013
C06184=1090.456,205.377,-72.567,176.273,20.045,153.013
C06185=1090.462,205.626,-72.591,176.276,20.046,153.013
C06186=1090.467,205.874,-72.615,176.279,20.047,153.012
C06187=1090.472,206.124,-72.639,176.281,20.048,153.012
C06188=1090.479,206.373,-72.663,176.284,20.050,153.012
C06189=1090.484,206.621,-72.687,176.287,20.051,153.012
C06190=1090.489,206.870,-72.711,176.291,20.052,153.011
C06191=1090.495,207.119,-72.734,176.293,20.053,153.011
C06192=1090.500,207.367,-72.758,176.296,20.054,153.011
C06193=1090.524,208.388,-72.857,176.362,20.087,153.007
C06194=1090.532,208.770,-72.894,176.367,20.090,153.007
C06195=1090.541,209.149,-72.931,176.371,20.093,153.006
C06196=1090.550,209.529,-72.968,176.375,20.096,153.006
C06197=1090.558,209.909,-73.006,176.380,20.099,153.006
C06198=1090.564,210.158,-73.030,176.383,20.101,153.006
C06199=1090.569,210.406,-73.055,176.385,20.103,153.006
C06200=1090.574,210.655,-73.079,176.388,20.106,153.006
C06201=1090.581,210.904,-73.103,176.391,20.108,153.006
C06202=1090.586,211.153,-73.127,176.394,20.110,153.006
C06203=1090.592,211.402,-73.152,176.397,20.112,153.006
C06204=1090.598,211.650,-73.177,176.400,20.114,153.006
C06205=1090.603,211.898,-73.201,176.402,20.116,153.006
C06206=1090.609,212.148,-73.226,176.405,20.118,153.006
C06207=1090.614,212.396,-73.250,176.408,20.120,153.006
C06208=1090.620,212.646,-73.274,176.411,20.122,153.006
C06209=1090.626,212.894,-73.299,176.414,20.124,153.006
C06210=1090.631,213.142,-73.324,176.416,20.126,153.006
C06211=1090.637,213.391,-73.348,176.419,20.128,153.006
C06212=1090.642,213.640,-73.373,176.422,20.130,153.006
C06213=1090.649,213.889,-73.398,176.425,20.132,153.006
C06214=1090.653,214.138,-73.423,176.427,20.134,153.006
C06215=1090.658,214.386,-73.447,176.431,20.136,153.006
C06216=1090.664,214.635,-73.472,176.433,20.138,153.006
C06217=1090.670,214.883,-73.497,176.436,20.140,153.006
C06218=1090.676,215.133,-73.521,176.439,20.142,153.006
C06219=1090.681,215.381,-73.545,176.442,20.145,153.006
C06220=1090.687,215.630,-73.571,176.444,20.146,153.006
C06221=1090.693,215.879,-73.595,176.448,20.149,153.006
C06222=1090.697,216.127,-73.620,176.450,20.151,153.006
C06223=1090.703,216.376,-73.645,176.453,20.153,153.005
C06224=1090.709,216.625,-73.670,176.456,20.155,153.006
C06225=1090.715,216.873,-73.695,176.459,20.157,153.005
C06226=1090.720,217.122,-73.719,176.461,20.159,153.005
C06227=1090.726,217.371,-73.744,176.464,20.161,153.005
C06228=1090.731,217.620,-73.769,176.467,20.163,153.005
C06229=1090.737,217.869,-73.794,176.470,20.165,153.005
C06230=1090.742,218.117,-73.819,176.473,20.167,153.005
C06231=1090.748,218.366,-73.844,176.476,20.169,153.005
C06232=1090.754,218.614,-73.868,176.478,20.171,153.005
C06233=1090.760,218.863,-73.893,176.482,20.173,153.005
C06234=1090.765,219.112,-73.919,176.484,20.175,153.005
C06235=1090.771,219.360,-73.944,176.487,20.177,153.005
C06236=1090.777,219.610,-73.969,176.490,20.179,153.005
C06237=1090.782,219.858,-73.994,176.493,20.182,153.005
C06238=1090.788,220.107,-74.019,176.495,20.183,153.005
C06239=1090.793,220.355,-74.044,176.499,20.186,153.005
C06240=1090.799,220.604,-74.068,176.501,20.188,153.005
C06241=1090.805,220.853,-74.094,176.504,20.190,153.005
C06242=1090.811,221.101,-74.119,176.507,20.192,153.005
C06243=1090.816,221.351,-74.144,176.510,20.194,153.005
C06244=1090.822,221.599,-74.169,176.512,20.196,153.005
C06245=1090.828,221.847,-74.194,176.516,20.198,153.005
C06246=1090.837,222.232,-74.233,176.520,20.201,153.005
C06247=1090.845,222.615,-74.272,176.525,20.205,153.005
C06248=1090.853,222.999,-74.310,176.529,20.208,153.005
C06249=1090.862,223.383,-74.350,176.534,20.211,153.005
C06250=1090.867,223.632,-74.375,176.536,20.213,153.005
C06251=1090.873,223.880,-74.401,176.539,20.216,153.005
C06252=1090.878,224.129,-74.426,176.542,20.217,153.005
C06253=1090.884,224.378,-74.451,176.545,20.220,153.005
C06254=1090.890,224.627,-74.476,176.547,20.222,153.005
C06255=1090.895,224.875,-74.502,176.550,20.224,153.005
C06256=1090.902,225.123,-74.527,176.553,20.226,153.005
C06257=1090.907,225.373,-74.552,176.556,20.228,153.004
C06258=1090.912,225.621,-74.577,176.559,20.230,153.004
C06259=1090.918,225.870,-74.603,176.562,20.232,153.004
C06260=1090.924,226.119,-74.629,176.565,20.234,153.004
C06261=1090.929,226.367,-74.654,176.567,20.236,153.004
C06262=1090.935,226.616,-74.679,176.571,20.239,153.004
C06263=1090.940,226.865,-74.705,176.573,20.240,153.004
C06264=1090.946,227.113,-74.730,176.576,20.243,153.004
C06265=1090.952,227.362,-74.756,176.579,20.245,153.004
C06266=1090.958,227.610,-74.782,176.582,20.247,153.004
C06267=1090.963,227.859,-74.807,176.584,20.249,153.004
C06268=1090.969,228.108,-74.832,176.588,20.251,153.004
C06269=1090.974,228.357,-74.858,176.591,20.253,153.004
C06270=1090.980,228.605,-74.883,176.593,20.255,153.004
C06271=1090.985,228.854,-74.909,176.597,20.257,153.004
C06272=1090.992,229.102,-74.935,176.599,20.259,153.004
C06273=1090.997,229.351,-74.961,176.602,20.261,153.004
C06274=1091.003,229.600,-74.987,176.605,20.263,153.004
C06275=1091.008,229.848,-75.012,176.608,20.266,153.004
C06276=1091.014,230.097,-75.037,176.611,20.268,153.004
C06277=1091.020,230.345,-75.063,176.614,20.270,153.004
C06278=1091.025,230.594,-75.089,176.617,20.272,153.004
C06279=1091.030,230.843,-75.114,176.619,20.274,153.004
C06280=1091.036,231.091,-75.140,176.623,20.276,153.004
C06281=1091.042,231.340,-75.166,176.625,20.278,153.004
C06282=1091.048,231.589,-75.192,176.628,20.280,153.004
C06283=1091.053,231.837,-75.217,176.631,20.283,153.004
C06284=1091.059,232.086,-75.243,176.634,20.285,153.004
C06285=1091.064,232.335,-75.269,176.637,20.287,153.004
C06286=1091.070,232.584,-75.295,176.639,20.289,153.004
C06287=1091.076,232.832,-75.320,176.643,20.291,153.004
C06288=1091.081,233.080,-75.347,176.646,20.294,153.004
C06289=1091.086,233.329,-75.373,176.648,20.295,153.004
C06290=1091.092,233.578,-75.398,176.652,20.298,153.004
C06291=1091.098,233.827,-75.424,176.654,20.300,153.004
C06292=1091.104,234.075,-75.450,176.657,20.302,153.004
C06293=1091.109,234.323,-75.476,176.660,20.305,153.004
C06294=1091.114,234.572,-75.502,176.663,20.307,153.004
C06295=1091.120,234.820,-75.529,176.666,20.309,153.004
C06296=1091.126,235.069,-75.554,176.669,20.311,153.004
C06297=1091.132,235.318,-75.580,176.672,20.313,153.004
C06298=1091.140,235.693,-75.620,176.677,20.317,153.004
C06299=1091.148,236.068,-75.659,176.681,20.320,153.004
C06300=1091.157,236.444,-75.698,176.685,20.323,153.004
C06301=1091.165,236.819,-75.738,176.690,20.326,153.004
C06302=1091.171,237.068,-75.764,176.693,20.329,153.004
C06303=1091.176,237.316,-75.790,176.695,20.330,153.004
C06304=1091.182,237.565,-75.817,176.698,20.333,153.004
C06305=1091.187,237.814,-75.843,176.701,20.335,153.004
C06306=1091.193,238.062,-75.869,176.704,20.337,153.004
C06307=1091.199,238.311,-75.894,176.707,20.339,153.003
C06308=1091.205,238.559,-75.921,176.710,20.341,153.004
C06309=1091.210,238.807,-75.947,176.713,20.344,153.004
C06310=1091.216,239.056,-75.973,176.716,20.346,153.003
C06311=1091.221,239.305,-75.999,176.719,20.348,153.003
C06312=1091.227,239.553,-76.026,176.722,20.350,153.003
C06313=1091.233,239.802,-76.053,176.724,20.352,153.003
C06314=1091.238,240.051,-76.079,176.728,20.354,153.003
C06315=1091.244,240.299,-76.105,176.731,20.357,153.003
C06316=1091.250,240.548,-76.131,176.733,20.359,153.003
C06317=1091.255,240.796,-76.158,176.736,20.361,153.003
C06318=1091.261,241.045,-76.184,176.740,20.363,153.003
C06319=1091.267,241.294,-76.210,176.742,20.365,153.003
C06320=1091.272,241.542,-76.237,176.745,20.367,153.003
C06321=1091.278,241.790,-76.264,176.749,20.370,153.003
C06322=1091.284,242.039,-76.290,176.751,20.372,153.003
C06323=1091.289,242.288,-76.316,176.754,20.374,153.003
C06324=1091.295,242.536,-76.343,176.757,20.376,153.003
C06325=1091.301,242.784,-76.369,176.760,20.378,153.003
C06326=1091.306,243.033,-76.395,176.763,20.381,153.003
C06327=1091.312,243.282,-76.422,176.766,20.383,153.003
C06328=1091.317,243.530,-76.449,176.769,20.385,153.003
C06329=1091.323,243.779,-76.476,176.772,20.387,153.003
C06330=1091.329,244.027,-76.503,176.775,20.390,153.003
C06331=1091.334,244.276,-76.529,176.777,20.392,153.003
C06332=1091.340,244.524,-76.555,176.781,20.394,153.003
C06333=1091.345,244.773,-76.582,176.784,20.396,153.003
C06334=1091.351,245.021,-76.609,176.786,20.398,153.003
C06335=1091.357,245.270,-76.636,176.789,20.401,153.003
C06336=1091.362,245.518,-76.662,176.793,20.403,153.003
C06337=1091.368,245.767,-76.689,176.795,20.405,153.003
C06338=1091.373,246.016,-76.716,176.798,20.407,153.003
C06339=1091.379,246.264,-76.742,176.802,20.410,153.003
C06340=1091.384,246.513,-76.769,176.804,20.412,153.003
C06341=1091.390,246.761,-76.796,176.807,20.414,153.003
C06342=1091.395,247.010,-76.823,176.810,20.416,153.003
C06343=1091.402,247.259,-76.850,176.813,20.418,153.003
C06344=1091.407,247.507,-76.876,176.816,20.421,153.003
C06345=1091.412,247.756,-76.904,176.819,20.423,153.003
C06346=1091.418,248.004,-76.930,176.822,20.426,153.003
C06347=1091.424,248.252,-76.957,176.825,20.428,153.003
C06348=1091.429,248.501,-76.984,176.828,20.430,153.003
C06349=1091.435,248.749,-77.011,176.831,20.432,153.003
C06350=1091.443,249.118,-77.051,176.835,20.436,153.003
C06351=1091.451,249.486,-77.091,176.840,20.439,153.003
C06352=1091.459,249.854,-77.131,176.844,20.442,153.003
C06353=1091.468,250.223,-77.171,176.849,20.446,153.004
C06354=1091.473,250.471,-77.198,176.851,20.448,153.004
C06355=1091.479,250.719,-77.225,176.854,20.450,153.003
C06356=1091.484,250.968,-77.253,176.858,20.453,153.003
C06357=1091.490,251.216,-77.279,176.860,20.455,153.004
C06358=1091.495,251.466,-77.307,176.863,20.457,153.004
C06359=1091.501,251.714,-77.333,176.866,20.460,153.004
C06360=1091.506,251.962,-77.361,176.869,20.462,153.004
C06361=1091.512,252.210,-77.388,176.872,20.464,153.004
C06362=1091.517,252.459,-77.415,176.875,20.467,153.004
C06363=1091.523,252.707,-77.442,176.878,20.469,153.004
C06364=1091.529,252.956,-77.470,176.882,20.471,153.004
C06365=1091.535,253.205,-77.497,176.884,20.473,153.004
C06366=1091.540,253.453,-77.524,176.887,20.476,153.004
C06367=1091.546,253.701,-77.552,176.890,20.478,153.004
C06368=1091.551,253.950,-77.579,176.893,20.480,153.004
C06369=1091.557,254.199,-77.606,176.896,20.483,153.004
C06370=1091.562,254.447,-77.634,176.899,20.485,153.004
C06371=1091.568,254.695,-77.660,176.902,20.488,153.004
C06372=1091.573,254.944,-77.688,176.905,20.489,153.004
C06373=1091.579,255.192,-77.716,176.908,20.492,153.004
C06374=1091.585,255.441,-77.743,176.911,20.494,153.004
C06375=1091.590,255.689,-77.771,176.914,20.497,153.004
C06376=1091.596,255.937,-77.797,176.917,20.499,153.004
C06377=1091.601,256.186,-77.825,176.920,20.501,153.004
C06378=1091.608,256.434,-77.852,176.923,20.504,153.004
C06379=1091.613,256.683,-77.879,176.926,20.506,153.004
C06380=1091.618,256.931,-77.907,176.929,20.508,153.004
C06381=1091.625,257.180,-77.934,176.932,20.510,153.004
C06382=1091.630,257.428,-77.962,176.935,20.513,153.004
C06383=1091.636,257.677,-77.989,176.938,20.515,153.004
C06384=1091.641,257.925,-78.017,176.941,20.517,153.004
C06385=1091.647,258.173,-78.045,176.944,20.520,153.004
C06386=1091.653,258.422,-78.072,176.947,20.522,153.004
C06387=1091.658,258.670,-78.100,176.950,20.524,153.004
C06388=1091.664,258.919,-78.127,176.953,20.526,153.004
C06389=1091.670,259.167,-78.155,176.956,20.529,153.004
C06390=1091.676,259.416,-78.183,176.959,20.531,153.004
C06391=1091.682,259.664,-78.210,176.962,20.534,153.004
C06392=1091.687,259.912,-78.238,176.965,20.536,153.004
C06393=1091.693,260.161,-78.266,176.968,20.538,153.004
C06394=1091.699,260.409,-78.293,176.971,20.540,153.004
C06395=1091.704,260.657,-78.321,176.974,20.543,153.004
C06396=1091.710,260.906,-78.349,176.978,20.545,153.004
C06397=1091.716,261.154,-78.376,176.980,20.547,153.004
C06398=1091.722,261.403,-78.404,176.983,20.550,153.004
C06399=1091.727,261.651,-78.432,176.986,20.552,153.004
C06400=1091.733,261.899,-78.459,176.990,20.555,153.004
C06401=1091.739,262.148,-78.487,176.992,20.557,153.004
C06402=1091.747,262.513,-78.528,176.997,20.560,153.004
C06403=1091.756,262.878,-78.569,177.002,20.564,153.004
C06404=1091.763,263.244,-78.610,177.006,20.567,153.004
C06405=1091.773,263.610,-78.651,177.010,20.571,153.004
C06406=1091.778,263.858,-78.679,177.014,20.573,153.004
C06407=1091.784,264.107,-78.708,177.016,20.575,153.004
C06408=1091.790,264.354,-78.735,177.019,20.577,153.004
C06409=1091.796,264.604,-78.763,177.022,20.580,153.004
C06410=1091.801,264.852,-78.791,177.026,20.582,153.004
C06411=1091.806,265.100,-78.819,177.029,20.585,153.004
C06412=1091.812,265.349,-78.847,177.031,20.586,153.004
C06413=1091.818,265.597,-78.875,177.034,20.589,153.004
C06414=1091.824,265.845,-78.903,177.038,20.591,153.005
C06415=1091.829,266.093,-78.931,177.041,20.594,153.005
C06416=1091.835,266.342,-78.959,177.044,20.596,153.005
C06417=1091.840,266.590,-78.987,177.046,20.598,153.005
C06418=1091.846,266.839,-79.016,177.050,20.601,153.005
C06419=1091.852,267.087,-79.044,177.052,20.604,153.005
C06420=1091.858,267.336,-79.072,177.056,20.606,153.005
C06421=1091.863,267.583,-79.101,177.059,20.609,153.005
C06422=1091.869,267.831,-79.129,177.061,20.611,153.005
C06423=1091.874,268.080,-79.157,177.064,20.613,153.005
C06424=1091.880,268.328,-79.185,177.068,20.616,153.005
C06425=1091.886,268.577,-79.213,177.071,20.618,153.005
C06426=1091.892,268.826,-79.242,177.074,20.621,153.005
C06427=1091.897,269.074,-79.270,177.077,20.623,153.005
C06428=1091.903,269.322,-79.298,177.079,20.625,153.005
C06429=1091.909,269.570,-79.327,177.083,20.628,153.005
C06430=1091.915,269.819,-79.355,177.086,20.630,153.005
C06431=1091.920,270.067,-79.383,177.089,20.633,153.005
C06432=1091.925,270.316,-79.412,177.092,20.635,153.005
C06433=1091.931,270.563,-79.440,177.095,20.638,153.005
C06434=1091.937,270.812,-79.469,177.098,20.640,153.005
C06435=1091.942,271.060,-79.497,177.101,20.642,153.005
C06436=1091.948,271.309,-79.525,177.104,20.645,153.006
C06437=1091.954,271.556,-79.554,177.107,20.648,153.006
C06438=1091.960,271.805,-79.582,177.110,20.650,153.006
C06439=1091.965,272.054,-79.611,177.114,20.653,153.006
C06440=1091.970,272.301,-79.640,177.117,20.655,153.006
C06441=1091.976,272.550,-79.668,177.119,20.657,153.006
C06442=1091.982,272.798,-79.696,177.122,20.660,153.006
C06443=1091.988,273.046,-79.725,177.125,20.662,153.006
C06444=1091.993,273.295,-79.754,177.128,20.665,153.006
C06445=1091.999,273.543,-79.783,177.132,20.668,153.006
C06446=1092.005,273.791,-79.811,177.135,20.670,153.006
C06447=1092.010,274.039,-79.840,177.138,20.672,153.006
C06448=1092.016,274.288,-79.868,177.140,20.674,153.006
C06449=1092.022,274.537,-79.897,177.144,20.677,153.006
C06450=1092.027,274.784,-79.925,177.147,20.680,153.006
C06451=1092.032,275.033,-79.954,177.150,20.682,153.006
C06452=1092.038,275.281,-79.983,177.153,20.685,153.006
C06453=1092.044,275.529,-80.011,177.156,20.687,153.007
C06454=1092.052,275.897,-80.055,177.161,20.691,153.007
C06455=1092.061,276.266,-80.098,177.165,20.695,153.007
C06456=1092.069,276.634,-80.140,177.170,20.698,153.007
C06457=1092.078,277.002,-80.183,177.174,20.702,153.007
C06458=1092.083,277.251,-80.212,177.177,20.705,153.007
C06459=1092.089,277.499,-80.241,177.180,20.708,153.007
C06460=1092.095,277.746,-80.269,177.183,20.710,153.007
C06461=1092.100,277.996,-80.298,177.186,20.712,153.007
C06462=1092.106,278.244,-80.327,177.189,20.715,153.007
C06463=1092.111,278.491,-80.357,177.192,20.718,153.007
C06464=1092.117,278.740,-80.385,177.195,20.720,153.007
C06465=1092.123,278.988,-80.414,177.198,20.723,153.007
C06466=1092.128,279.236,-80.443,177.202,20.725,153.008
C06467=1092.134,279.484,-80.472,177.205,20.728,153.008
C06468=1092.140,279.733,-80.501,177.208,20.730,153.008
C06469=1092.146,279.981,-80.530,177.211,20.733,153.008
C06470=1092.151,280.229,-80.560,177.213,20.735,153.008
C06471=1092.157,280.477,-80.589,177.216,20.738,153.008
C06472=1092.163,280.726,-80.618,177.220,20.740,153.008
C06473=1092.169,280.974,-80.647,177.223,20.743,153.008
C06474=1092.173,281.222,-80.676,177.226,20.746,153.008
C06475=1092.180,281.470,-80.705,177.229,20.748,153.008
C06476=1092.185,281.719,-80.734,177.232,20.751,153.008
C06477=1092.191,281.967,-80.764,177.235,20.754,153.008
C06478=1092.196,282.215,-80.793,177.238,20.756,153.009
C06479=1092.202,282.463,-80.822,177.241,20.759,153.009
C06480=1092.208,282.711,-80.851,177.244,20.762,153.009
C06481=1092.214,282.960,-80.881,177.248,20.764,153.009
C06482=1092.219,283.207,-80.910,177.251,20.767,153.009
C06483=1092.225,283.455,-80.939,177.253,20.769,153.009
C06484=1092.230,283.704,-80.969,177.256,20.772,153.009
C06485=1092.236,283.952,-80.999,177.259,20.774,153.009
C06486=1092.242,284.201,-81.028,177.262,20.777,153.009
C06487=1092.247,284.448,-81.057,177.265,20.780,153.009
C06488=1092.252,284.697,-81.087,177.269,20.782,153.010
C06489=1092.259,284.945,-81.116,177.272,20.785,153.010
C06490=1092.264,285.193,-81.145,177.275,20.788,153.010
C06491=1092.270,285.442,-81.175,177.278,20.790,153.010
C06492=1092.276,285.690,-81.204,177.281,20.793,153.010
C06493=1092.281,285.938,-81.233,177.284,20.796,153.010
C06494=1092.286,286.186,-81.263,177.287,20.798,153.010
C06495=1092.292,286.434,-81.293,177.290,20.801,153.010
C06496=1092.299,286.682,-81.322,177.293,20.804,153.010
C06497=1092.304,286.930,-81.352,177.296,20.807,153.010
C06498=1092.310,287.179,-81.382,177.300,20.809,153.010
C06499=1092.315,287.427,-81.411,177.303,20.812,153.011
C06500=1092.321,287.674,-81.441,177.306,20.815,153.011
C06501=1092.327,287.923,-81.470,177.309,20.817,153.011
C06502=1092.332,288.171,-81.500,177.311,20.819,153.011
C06503=1092.338,288.419,-81.529,177.314,20.822,153.011
C06504=1092.344,288.667,-81.559,177.317,20.825,153.011
C06505=1092.350,288.915,-81.589,177.321,20.827,153.011
C06506=1092.358,289.293,-81.634,177.325,20.831,153.011
C06507=1092.367,289.671,-81.679,177.330,20.836,153.012
C06508=1092.376,290.049,-81.724,177.335,20.840,153.012
C06509=1092.384,290.426,-81.770,177.340,20.844,153.012
C06510=1092.390,290.674,-81.800,177.343,20.847,153.012
C06511=1092.395,290.922,-81.830,177.346,20.850,153.012
C06512=1092.401,291.171,-81.859,177.349,20.852,153.012
C06513=1092.407,291.418,-81.889,177.352,20.855,153.012
C06514=1092.412,291.667,-81.919,177.355,20.858,153.012
C06515=1092.418,291.915,-81.949,177.358,20.861,153.013
C06516=1092.423,292.163,-81.979,177.362,20.863,153.013
C06517=1092.429,292.411,-82.009,177.365,20.866,153.013
C06518=1092.435,292.659,-82.039,177.368,20.869,153.013
C06519=1092.441,292.907,-82.069,177.371,20.872,153.013
C06520=1092.446,293.156,-82.099,177.374,20.875,153.013
C06521=1092.452,293.404,-82.129,177.377,20.877,153.013
C06522=1092.458,293.651,-82.160,177.380,20.880,153.013
C06523=1092.463,293.900,-82.189,177.383,20.883,153.014
C06524=1092.469,294.148,-82.220,177.386,20.885,153.014
C06525=1092.475,294.396,-82.249,177.389,20.888,153.014
C06526=1092.480,294.644,-82.280,177.392,20.891,153.014
C06527=1092.486,294.892,-82.310,177.395,20.894,153.014
C06528=1092.492,295.140,-82.340,177.398,20.897,153.014
C06529=1092.498,295.388,-82.370,177.401,20.899,153.014
C06530=1092.503,295.636,-82.400,177.404,20.902,153.015
C06531=1092.509,295.884,-82.430,177.407,20.905,153.015
C06532=1092.515,296.132,-82.460,177.411,20.908,153.015
C06533=1092.521,296.380,-82.491,177.414,20.911,153.015
C06534=1092.526,296.628,-82.521,177.417,20.913,153.015
C06535=1092.532,296.877,-82.552,177.420,20.916,153.015
C06536=1092.538,297.125,-82.582,177.423,20.919,153.015
C06537=1092.543,297.373,-82.612,177.426,20.922,153.016
C06538=1092.549,297.621,-82.643,177.429,20.925,153.016
C06539=1092.555,297.869,-82.672,177.432,20.927,153.016
C06540=1092.561,298.117,-82.703,177.435,20.930,153.016
C06541=1092.566,298.365,-82.734,177.438,20.933,153.016
C06542=1092.571,298.613,-82.764,177.441,20.936,153.016
C06543=1092.577,298.861,-82.794,177.444,20.939,153.017
C06544=1092.582,299.109,-82.825,177.447,20.942,153.017
C06545=1092.588,299.357,-82.856,177.450,20.945,153.017
C06546=1092.594,299.604,-82.886,177.454,20.948,153.017
C06547=1092.599,299.853,-82.917,177.457,20.951,153.017
C06548=1092.605,300.101,-82.947,177.460,20.954,153.017
C06549=1092.610,300.349,-82.978,177.463,20.957,153.017
C06550=1092.616,300.598,-83.008,177.466,20.960,153.018
C06551=1092.622,300.845,-83.039,177.469,20.963,153.018
C06552=1092.627,301.094,-83.070,177.472,20.965,153.018
C06553=1092.633,301.341,-83.100,177.475,20.968,153.018
C06554=1092.638,301.590,-83.131,177.478,20.971,153.018
C06555=1092.644,301.837,-83.162,177.481,20.974,153.019
C06556=1092.650,302.085,-83.192,177.484,20.977,153.019
C06557=1092.655,302.333,-83.223,177.487,20.980,153.019
C06558=1092.664,302.725,-83.271,177.492,20.985,153.019
C06559=1092.673,303.116,-83.320,177.497,20.989,153.019
C06560=1092.682,303.508,-83.369,177.502,20.994,153.020
C06561=1092.691,303.900,-83.418,177.507,20.999,153.020
C06562=1092.696,304.147,-83.448,177.510,21.002,153.020
C06563=1092.702,304.396,-83.479,177.513,21.005,153.020
C06564=1092.707,304.643,-83.509,177.516,21.008,153.021
C06565=1092.713,304.892,-83.541,177.519,21.011,153.021
C06566=1092.719,305.139,-83.572,177.522,21.014,153.021
C06567=1092.724,305.388,-83.603,177.525,21.017,153.021
C06568=1092.730,305.635,-83.633,177.528,21.020,153.021
C06569=1092.736,305.884,-83.665,177.531,21.023,153.021
C06570=1092.742,306.131,-83.695,177.534,21.026,153.022
C06571=1092.747,306.380,-83.726,177.537,21.029,153.022
C06572=1092.753,306.627,-83.758,177.541,21.032,153.022
C06573=1092.759,306.876,-83.789,177.544,21.035,153.022
C06574=1092.765,307.123,-83.819,177.547,21.038,153.023
C06575=1092.770,307.371,-83.851,177.550,21.041,153.023
C06576=1092.776,307.619,-83.881,177.553,21.044,153.023
C06577=1092.782,307.867,-83.913,177.556,21.047,153.023
C06578=1092.787,308.115,-83.944,177.559,21.050,153.023
C06579=1092.793,308.363,-83.975,177.562,21.053,153.023
C06580=1092.799,308.611,-84.007,177.566,21.056,153.024
C06581=1092.804,308.859,-84.037,177.569,21.059,153.024
C06582=1092.810,309.106,-84.069,177.572,21.062,153.024
C06583=1092.816,309.355,-84.099,177.575,21.065,153.024
C06584=1092.822,309.602,-84.131,177.578,21.068,153.024
C06585=1092.827,309.851,-84.162,177.581,21.071,153.025
C06586=1092.833,310.098,-84.193,177.584,21.074,153.025
C06587=1092.839,310.347,-84.224,177.588,21.078,153.025
C06588=1092.845,310.595,-84.256,177.591,21.081,153.025
C06589=1092.851,310.842,-84.287,177.594,21.084,153.025
C06590=1092.856,311.091,-84.319,177.597,21.087,153.026
C06591=1092.862,311.338,-84.350,177.600,21.090,153.026
C06592=1092.868,311.586,-84.381,177.602,21.093,153.026
C06593=1092.873,311.834,-84.413,177.606,21.096,153.026
C06594=1092.880,312.082,-84.444,177.609,21.099,153.027
C06595=1092.885,312.330,-84.475,177.612,21.102,153.027
C06596=1092.891,312.578,-84.507,177.615,21.105,153.027
C06597=1092.897,312.826,-84.538,177.618,21.108,153.027
C06598=1092.903,313.073,-84.570,177.621,21.111,153.027
C06599=1092.908,313.322,-84.601,177.624,21.114,153.028
C06600=1092.914,313.570,-84.633,177.628,21.118,153.028
C06601=1092.921,313.818,-84.664,177.631,21.121,153.028
C06602=1092.926,314.065,-84.696,177.634,21.124,153.028
C06603=1092.932,314.314,-84.727,177.637,21.127,153.029
C06604=1092.938,314.561,-84.758,177.640,21.130,153.029
C06605=1092.944,314.809,-84.790,177.644,21.133,153.029
C06606=1092.949,315.057,-84.822,177.647,21.136,153.029
C06607=1092.955,315.305,-84.854,177.649,21.140,153.029
C06608=1092.960,315.553,-84.885,177.652,21.143,153.030
C06609=1092.966,315.801,-84.917,177.655,21.146,153.030
C06610=1092.975,316.195,-84.968,177.660,21.151,153.030
C06611=1092.984,316.590,-85.018,177.665,21.157,153.031
C06612=1092.993,316.984,-85.069,177.670,21.162,153.031
C06613=1093.002,317.379,-85.119,177.675,21.167,153.032
C06614=1093.007,317.626,-85.151,177.678,21.170,153.032
C06615=1093.013,317.874,-85.183,177.681,21.173,153.032
C06616=1093.019,318.122,-85.215,177.684,21.177,153.032
C06617=1093.025,318.370,-85.247,177.687,21.180,153.033
C06618=1093.029,318.618,-85.279,177.690,21.183,153.033
C06619=1093.035,318.866,-85.311,177.693,21.187,153.033
C06620=1093.041,319.113,-85.343,177.697,21.190,153.033
C06621=1093.047,319.361,-85.375,177.700,21.194,153.034
C06622=1093.052,319.609,-85.407,177.702,21.197,153.034
C06623=1093.058,319.857,-85.439,177.705,21.200,153.034
C06624=1093.064,320.105,-85.471,177.708,21.203,153.035
C06625=1093.069,320.353,-85.503,177.712,21.207,153.035
C06626=1093.075,320.601,-85.535,177.715,21.210,153.035
C06627=1093.080,320.849,-85.567,177.718,21.213,153.035
C06628=1093.086,321.096,-85.600,177.720,21.217,153.036
C06629=1093.092,321.344,-85.631,177.724,21.221,153.036
C06630=1093.098,321.592,-85.663,177.727,21.224,153.036
C06631=1093.103,321.841,-85.696,177.730,21.227,153.037
C06632=1093.109,322.087,-85.728,177.733,21.230,153.037
C06633=1093.115,322.336,-85.760,177.737,21.234,153.037
C06634=1093.121,322.584,-85.792,177.739,21.237,153.037
C06635=1093.126,322.831,-85.824,177.742,21.240,153.038
C06636=1093.132,323.079,-85.857,177.745,21.244,153.038
C06637=1093.138,323.327,-85.889,177.749,21.247,153.038
C06638=1093.143,323.575,-85.921,177.752,21.251,153.039
C06639=1093.149,323.823,-85.954,177.755,21.254,153.039
C06640=1093.155,324.071,-85.986,177.757,21.257,153.039
C06641=1093.160,324.319,-86.018,177.761,21.261,153.040
C06642=1093.166,324.566,-86.051,177.764,21.264,153.040
C06643=1093.172,324.814,-86.083,177.767,21.268,153.040
C06644=1093.178,325.062,-86.116,177.770,21.271,153.040
C06645=1093.183,325.310,-86.148,177.773,21.275,153.041
C06646=1093.190,325.557,-86.181,177.776,21.278,153.041
C06647=1093.195,325.806,-86.213,177.779,21.281,153.042
C06648=1093.201,326.054,-86.246,177.783,21.285,153.042
C06649=1093.206,326.301,-86.278,177.786,21.288,153.042
C06650=1093.213,326.549,-86.310,177.788,21.292,153.042
C06651=1093.218,326.797,-86.343,177.792,21.296,153.043
C06652=1093.224,327.045,-86.376,177.795,21.299,153.043
C06653=1093.230,327.292,-86.407,177.798,21.302,153.043
C06654=1093.235,327.540,-86.441,177.800,21.306,153.044
C06655=1093.241,327.788,-86.473,177.804,21.309,153.044
C06656=1093.247,328.036,-86.506,177.807,21.313,153.044
C06657=1093.253,328.284,-86.539,177.810,21.316,153.045
C06658=1093.259,328.532,-86.571,177.814,21.320,153.045
C06659=1093.264,328.779,-86.604,177.816,21.323,153.045
C06660=1093.270,329.027,-86.637,177.819,21.326,153.046
C06661=1093.276,329.275,-86.669,177.823,21.330,153.046
C06662=1093.286,329.662,-86.720,177.827,21.336,153.046
C06663=1093.295,330.050,-86.771,177.832,21.341,153.047
C06664=1093.304,330.437,-86.822,177.837,21.347,153.047
C06665=1093.313,330.824,-86.874,177.842,21.352,153.048
C06666=1093.319,331.072,-86.907,177.845,21.356,153.048
C06667=1093.325,331.320,-86.940,177.848,21.359,153.049
C06668=1093.330,331.568,-86.973,177.851,21.363,153.049
C06669=1093.336,331.816,-87.005,177.854,21.366,153.049
C06670=1093.343,332.064,-87.038,177.857,21.370,153.050
C06671=1093.348,332.311,-87.071,177.861,21.374,153.050
C06672=1093.353,332.559,-87.104,177.863,21.377,153.050
C06673=1093.360,332.806,-87.137,177.867,21.381,153.051
C06674=1093.365,333.054,-87.170,177.870,21.385,153.051
C06675=1093.371,333.302,-87.204,177.872,21.388,153.052
C06676=1093.377,333.550,-87.237,177.876,21.392,153.052
C06677=1093.383,333.798,-87.270,177.879,21.396,153.052
C06678=1093.388,334.046,-87.303,177.882,21.399,153.053
C06679=1093.394,334.293,-87.337,177.885,21.403,153.053
C06680=1093.400,334.541,-87.369,177.888,21.407,153.053
C06681=1093.405,334.788,-87.402,177.891,21.411,153.054
C06682=1093.410,335.036,-87.436,177.894,21.414,153.054
C06683=1093.417,335.284,-87.468,177.897,21.418,153.055
C06684=1093.422,335.532,-87.502,177.901,21.422,153.055
C06685=1093.428,335.780,-87.535,177.903,21.426,153.055
C06686=1093.433,336.027,-87.568,177.907,21.430,153.056
C06687=1093.440,336.275,-87.601,177.909,21.433,153.056
C06688=1093.445,336.523,-87.634,177.912,21.437,153.057
C06689=1093.451,336.771,-87.668,177.916,21.441,153.057
C06690=1093.457,337.018,-87.702,177.919,21.444,153.057
C06691=1093.463,337.266,-87.735,177.922,21.449,153.058
C06692=1093.469,337.514,-87.768,177.925,21.452,153.058
C06693=1093.474,337.762,-87.801,177.928,21.456,153.059
C06694=1093.480,338.009,-87.835,177.931,21.460,153.059
C06695=1093.485,338.257,-87.869,177.934,21.464,153.059
C06696=1093.492,338.504,-87.901,177.937,21.467,153.060
C06697=1093.497,338.752,-87.935,177.940,21.471,153.060
C06698=1093.503,338.999,-87.969,177.944,21.476,153.061
C06699=1093.509,339.247,-88.002,177.946,21.479,153.061
C06700=1093.514,339.495,-88.035,177.950,21.483,153.061
C06701=1093.520,339.743,-88.069,177.952,21.487,153.062
C06702=1093.526,339.991,-88.103,177.956,21.491,153.062
C06703=1093.532,340.239,-88.137,177.959,21.495,153.063
C06704=1093.538,340.486,-88.171,177.961,21.498,153.063
C06705=1093.543,340.734,-88.204,177.965,21.503,153.064
C06706=1093.549,340.982,-88.238,177.968,21.507,153.064
C06707=1093.555,341.229,-88.271,177.971,21.510,153.064
C06708=1093.561,341.477,-88.305,177.974,21.514,153.065
C06709=1093.566,341.725,-88.339,177.977,21.519,153.065
C06710=1093.572,341.972,-88.373,177.980,21.522,153.066
C06711=1093.578,342.220,-88.406,177.983,21.527,153.066
C06712=1093.583,342.467,-88.440,177.986,21.530,153.067
C06713=1093.589,342.715,-88.473,177.990,21.534,153.067
C06714=1093.598,343.096,-88.526,177.995,21.540,153.068
C06715=1093.607,343.478,-88.578,177.999,21.547,153.069
C06716=1093.616,343.859,-88.630,178.003,21.552,153.069
C06717=1093.625,344.241,-88.682,178.008,21.559,153.070
C06718=1093.631,344.488,-88.716,178.011,21.563,153.071
C06719=1093.637,344.737,-88.750,178.014,21.567,153.071
C06720=1093.642,344.984,-88.784,178.018,21.571,153.071
C06721=1093.648,345.231,-88.818,178.020,21.575,153.072
C06722=1093.654,345.479,-88.852,178.024,21.580,153.072
C06723=1093.660,345.727,-88.886,178.027,21.584,153.073
C06724=1093.665,345.974,-88.920,178.030,21.588,153.073
C06725=1093.671,346.222,-88.955,178.033,21.592,153.074
C06726=1093.677,346.469,-88.989,178.036,21.596,153.074
C06727=1093.683,346.717,-89.022,178.039,21.600,153.075
C06728=1093.688,346.965,-89.056,178.042,21.604,153.075
C06729=1093.694,347.212,-89.090,178.045,21.609,153.076
C06730=1093.700,347.460,-89.125,178.048,21.612,153.076
C06731=1093.706,347.708,-89.159,178.051,21.617,153.077
C06732=1093.712,347.955,-89.194,178.054,21.621,153.077
C06733=1093.717,348.202,-89.228,178.057,21.625,153.078
C06734=1093.723,348.450,-89.262,178.061,21.629,153.078
C06735=1093.729,348.698,-89.297,178.063,21.634,153.079
C06736=1093.735,348.945,-89.331,178.067,21.638,153.079
C06737=1093.740,349.193,-89.365,178.069,21.642,153.080
C06738=1093.746,349.440,-89.399,178.073,21.646,153.081
C06739=1093.752,349.688,-89.434,178.075,21.650,153.081
C06740=1093.758,349.935,-89.468,178.079,21.655,153.082
C06741=1093.763,350.183,-89.503,178.082,21.659,153.082
C06742=1093.769,350.431,-89.538,178.085,21.663,153.083
C06743=1093.775,350.678,-89.572,178.088,21.668,153.083
C06744=1093.781,350.926,-89.606,178.091,21.672,153.084
C06745=1093.786,351.173,-89.640,178.094,21.676,153.084
C06746=1093.792,351.421,-89.675,178.097,21.680,153.085
C06747=1093.798,351.668,-89.709,178.100,21.685,153.085
C06748=1093.803,351.916,-89.743,178.103,21.689,153.086
C06749=1093.810,352.163,-89.779,178.106,21.693,153.086
C06750=1093.815,352.411,-89.813,178.109,21.698,153.087
C06751=1093.821,352.658,-89.847,178.112,21.702,153.088
C06752=1093.828,352.906,-89.882,178.115,21.707,153.088
C06753=1093.833,353.154,-89.916,178.119,21.711,153.089
C06754=1093.840,353.401,-89.951,178.121,21.715,153.089
C06755=1093.845,353.649,-89.986,178.124,21.720,153.090
C06756=1093.850,353.896,-90.021,178.128,21.725,153.090
C06757=1093.857,354.144,-90.056,178.130,21.728,153.091
C06758=1093.862,354.391,-90.091,178.134,21.733,153.092
C06759=1093.868,354.639,-90.125,178.137,21.738,153.092
C06760=1093.874,354.886,-90.160,178.139,21.742,153.093
C06761=1093.879,355.134,-90.194,178.143,21.747,153.093
C06762=1093.885,355.381,-90.229,178.145,21.751,153.094
C06763=1093.891,355.629,-90.265,178.148,21.756,153.095
C06764=1093.896,355.876,-90.299,178.152,21.760,153.095
C06765=1093.903,356.124,-90.335,178.154,21.764,153.096
C06766=1093.911,356.508,-90.388,178.160,21.772,153.097
C06767=1093.921,356.892,-90.442,178.164,21.779,153.098
C06768=1093.930,357.275,-90.497,178.168,21.786,153.099
C06769=1093.938,357.660,-90.551,178.173,21.792,153.099
C06770=1093.944,357.907,-90.586,178.176,21.797,153.100
C06771=1093.951,358.154,-90.621,178.180,21.802,153.101
C06772=1093.956,358.402,-90.656,178.182,21.807,153.101
C06773=1093.962,358.649,-90.692,178.185,21.811,153.102
C06774=1093.967,358.896,-90.727,178.189,21.816,153.103
C06775=1093.974,359.144,-90.761,178.192,21.821,153.103
C06776=1093.979,359.391,-90.797,178.194,21.825,153.104
C06777=1093.985,359.639,-90.832,178.198,21.830,153.104
C06778=1093.991,359.886,-90.867,178.201,21.834,153.105
C06779=1093.997,360.134,-90.902,178.203,21.839,153.106
C06780=1094.002,360.381,-90.938,178.207,21.844,153.106
C06781=1094.008,360.629,-90.973,178.210,21.848,153.107
C06782=1094.014,360.876,-91.008,178.212,21.853,153.108
C06783=1094.020,361.123,-91.043,178.216,21.858,153.108
C06784=1094.026,361.370,-91.079,178.219,21.863,153.109
C06785=1094.032,361.618,-91.114,178.222,21.868,153.110
C06786=1094.037,361.865,-91.150,178.224,21.872,153.110
C06787=1094.043,362.113,-91.185,178.228,21.877,153.111
C06788=1094.048,362.360,-91.220,178.231,21.882,153.112
C06789=1094.054,362.608,-91.256,178.234,21.887,153.112
C06790=1094.061,362.855,-91.290,178.237,21.891,153.113
C06791=1094.067,363.102,-91.326,178.240,21.896,153.114
C06792=1094.073,363.350,-91.362,178.243,21.901,153.114
C06793=1094.078,363.597,-91.397,178.246,21.906,153.115
C06794=1094.084,363.845,-91.433,178.248,21.911,153.116
C06795=1094.090,364.092,-91.468,178.252,21.916,153.117
C06796=1094.096,364.339,-91.504,178.255,21.921,153.117
C06797=1094.102,364.587,-91.540,178.258,21.926,153.118
C06798=1094.107,364.834,-91.575,178.260,21.930,153.119
C06799=1094.113,365.082,-91.611,178.264,21.935,153.119
C06800=1094.119,365.329,-91.646,178.267,21.940,153.120
C06801=1094.125,365.576,-91.682,178.270,21.945,153.121
C06802=1094.131,365.823,-91.718,178.273,21.950,153.122
C06803=1094.136,366.070,-91.754,178.275,21.955,153.122
C06804=1094.142,366.318,-91.790,178.279,21.960,153.123
C06805=1094.148,366.566,-91.825,178.282,21.965,153.124
C06806=1094.154,366.813,-91.861,178.285,21.970,153.125
C06807=1094.160,367.060,-91.896,178.288,21.975,153.125
C06808=1094.166,367.307,-91.932,178.290,21.980,153.126
C06809=1094.171,367.555,-91.969,178.293,21.985,153.127
C06810=1094.177,367.802,-92.005,178.297,21.990,153.128
C06811=1094.183,368.049,-92.041,178.300,21.996,153.128
C06812=1094.189,368.296,-92.076,178.303,22.001,153.129
C06813=1094.195,368.544,-92.112,178.305,22.006,153.130
C06814=1094.200,368.790,-92.148,178.308,22.011,153.131
C06815=1094.206,369.038,-92.184,178.311,22.016,153.131
C06816=1094.212,369.286,-92.220,178.314,22.021,153.132
C06817=1094.218,369.533,-92.257,178.318,22.026,153.133
C06818=1094.227,369.932,-92.315,178.323,22.035,153.134
C06819=1094.237,370.331,-92.373,178.326,22.043,153.136
C06820=1094.246,370.731,-92.431,178.331,22.051,153.137
C06821=1094.255,371.130,-92.489,178.336,22.060,153.138
C06822=1094.262,371.377,-92.526,178.340,22.065,153.139
C06823=1094.267,371.624,-92.561,178.342,22.071,153.140
C06824=1094.273,371.871,-92.598,178.346,22.076,153.140
C06825=1094.279,372.119,-92.634,178.349,22.081,153.141
C06826=1094.285,372.366,-92.670,178.351,22.086,153.142
C06827=1094.291,372.613,-92.707,178.354,22.091,153.143
C06828=1094.296,372.860,-92.743,178.357,22.097,153.144
C06829=1094.302,373.107,-92.779,178.360,22.102,153.145
C06830=1094.309,373.354,-92.816,178.363,22.107,153.145
C06831=1094.314,373.602,-92.852,178.366,22.113,153.146
C06832=1094.320,373.849,-92.888,178.369,22.118,153.147
C06833=1094.327,374.096,-92.925,178.372,22.124,153.148
C06834=1094.331,374.344,-92.961,178.375,22.129,153.149
C06835=1094.338,374.591,-92.997,178.378,22.135,153.150
C06836=1094.343,374.838,-93.034,178.380,22.140,153.151
C06837=1094.350,375.085,-93.071,178.383,22.145,153.151
C06838=1094.355,375.333,-93.108,178.386,22.151,153.152
C06839=1094.361,375.579,-93.144,178.389,22.156,153.153
C06840=1094.366,375.827,-93.180,178.392,22.162,153.154
C06841=1094.373,376.074,-93.217,178.395,22.167,153.155
C06842=1094.378,376.321,-93.254,178.398,22.173,153.156
C06843=1094.385,376.568,-93.290,178.401,22.179,153.157
C06844=1094.390,376.816,-93.327,178.404,22.184,153.158
C06845=1094.396,377.063,-93.364,178.407,22.190,153.158
C06846=1094.401,377.309,-93.400,178.410,22.195,153.159
C06847=1094.408,377.556,-93.437,178.413,22.201,153.160
C06848=1094.413,377.804,-93.474,178.416,22.207,153.161
C06849=1094.419,378.051,-93.511,178.419,22.212,153.162
C06850=1094.425,378.298,-93.547,178.422,22.218,153.163
C06851=1094.431,378.546,-93.584,178.425,22.224,153.164
C06852=1094.437,378.793,-93.621,178.428,22.229,153.165
C06853=1094.443,379.040,-93.658,178.431,22.235,153.166
C06854=1094.449,379.287,-93.694,178.434,22.241,153.167
C06855=1094.455,379.534,-93.731,178.437,22.246,153.168
C06856=1094.461,379.781,-93.769,178.439,22.252,153.169
C06857=1094.467,380.028,-93.805,178.442,22.258,153.170
C06858=1094.472,380.275,-93.842,178.445,22.263,153.170
C06859=1094.478,380.522,-93.879,178.448,22.269,153.171
C06860=1094.484,380.769,-93.916,178.451,22.275,153.172
C06861=1094.490,381.016,-93.953,178.454,22.281,153.173
C06862=1094.496,381.263,-93.990,178.457,22.287,153.174
C06863=1094.502,381.510,-94.027,178.460,22.293,153.175
C06864=1094.507,381.758,-94.064,178.463,22.299,153.176
C06865=1094.514,382.005,-94.102,178.466,22.304,153.177
C06866=1094.520,382.252,-94.138,178.469,22.310,153.178
C06867=1094.526,382.500,-94.175,178.471,22.316,153.179
C06868=1094.532,382.746,-94.213,178.474,22.322,153.180
C06869=1094.537,382.994,-94.250,178.477,22.328,153.181
C06870=1094.543,383.206,-94.282,178.480,22.333,153.182
C06871=1094.548,383.420,-94.315,178.482,22.338,153.183
C06872=1094.552,383.633,-94.346,178.484,22.343,153.184
C06873=1094.557,383.847,-94.379,178.487,22.349,153.185
C06874=1094.563,384.060,-94.411,178.490,22.354,153.186
C06875=1094.568,384.272,-94.443,178.492,22.359,153.186
C06876=1094.573,384.486,-94.476,178.495,22.364,153.187
C06877=1094.578,384.700,-94.508,178.497,22.370,153.188
C06878=1094.584,384.947,-94.545,178.500,22.376,153.189
C06879=1094.589,385.194,-94.583,178.503,22.381,153.190
C06880=1094.595,385.441,-94.620,178.506,22.388,153.191
C06881=1094.602,385.687,-94.657,178.509,22.394,153.192
C06882=1094.607,385.935,-94.694,178.512,22.400,153.193
C06883=1094.613,386.181,-94.732,178.515,22.406,153.194
C06884=1094.619,386.429,-94.769,178.517,22.413,153.196
C06885=1094.625,386.676,-94.807,178.520,22.419,153.197
C06886=1094.631,386.922,-94.845,178.523,22.425,153.198
C06887=1094.637,387.169,-94.883,178.526,22.431,153.199
C06888=1094.642,387.416,-94.920,178.529,22.438,153.200
C06889=1094.649,387.664,-94.958,178.532,22.444,153.201
C06890=1094.655,387.911,-94.995,178.535,22.450,153.202
C06891=1094.661,388.157,-95.033,178.537,22.456,153.203
C06892=1094.666,388.405,-95.070,178.540,22.463,153.204
C06893=1094.672,388.651,-95.108,178.543,22.469,153.205
C06894=1094.678,388.898,-95.146,178.546,22.476,153.207
C06895=1094.684,389.146,-95.184,178.549,22.482,153.208
C06896=1094.690,389.392,-95.222,178.552,22.488,153.209
C06897=1094.696,389.639,-95.259,178.555,22.494,153.210
C06898=1094.702,389.886,-95.297,178.557,22.501,153.211
C06899=1094.708,390.133,-95.335,178.560,22.507,153.212
C06900=1094.714,390.381,-95.372,178.564,22.514,153.213
C06901=1094.719,390.628,-95.411,178.566,22.520,153.214
C06902=1094.725,390.874,-95.448,178.569,22.527,153.216
C06903=1094.731,391.121,-95.486,178.572,22.533,153.217
C06904=1094.738,391.369,-95.524,178.575,22.540,153.218
C06905=1094.744,391.615,-95.562,178.578,22.546,153.219
C06906=1094.750,391.861,-95.601,178.581,22.553,153.220
C06907=1094.756,392.109,-95.639,178.583,22.559,153.221
C06908=1094.762,392.356,-95.676,178.586,22.565,153.222
C06909=1094.767,392.603,-95.715,178.589,22.573,153.224
C06910=1094.774,392.850,-95.753,178.592,22.579,153.225
C06911=1094.780,393.097,-95.791,178.595,22.586,153.226
C06912=1094.786,393.344,-95.828,178.597,22.592,153.227
C06913=1094.792,393.591,-95.867,178.601,22.599,153.228
C06914=1094.798,393.838,-95.906,178.603,22.606,153.230
C06915=1094.804,394.084,-95.943,178.606,22.612,153.231
C06916=1094.809,394.332,-95.982,178.608,22.619,153.232
C06917=1094.815,394.579,-96.020,178.612,22.626,153.233
C06918=1094.822,394.825,-96.058,178.614,22.633,153.235
C06919=1094.827,395.073,-96.097,178.617,22.640,153.236
C06920=1094.833,395.319,-96.135,178.620,22.646,153.237
C06921=1094.838,395.566,-96.173,178.623,22.654,153.238
C06922=1094.845,395.813,-96.212,178.626,22.660,153.240
C06923=1094.851,396.060,-96.250,178.628,22.667,153.241
C06924=1094.857,396.307,-96.289,178.631,22.674,153.242
C06925=1094.863,396.554,-96.327,178.634,22.681,153.244
C06926=1094.868,396.774,-96.361,178.637,22.688,153.245
C06927=1094.873,396.993,-96.396,178.639,22.693,153.246
C06928=1094.878,397.213,-96.430,178.641,22.700,153.247
C06929=1094.883,397.433,-96.464,178.644,22.706,153.248
C06930=1094.889,397.653,-96.499,178.647,22.712,153.249
C06931=1094.895,397.872,-96.533,178.649,22.718,153.250
C06932=1094.900,398.092,-96.567,178.651,22.725,153.252
C06933=1094.905,398.312,-96.601,178.654,22.731,153.253
C06934=1094.911,398.559,-96.640,178.656,22.738,153.254
C06935=1094.918,398.805,-96.679,178.660,22.745,153.255
C06936=1094.923,399.053,-96.718,178.662,22.753,153.257
C06937=1094.929,399.299,-96.756,178.665,22.760,153.258
C06938=1094.935,399.547,-96.795,178.668,22.767,153.259
C06939=1094.941,399.793,-96.834,178.670,22.774,153.261
C06940=1094.948,400.040,-96.873,178.673,22.781,153.262
C06941=1094.953,400.287,-96.911,178.676,22.789,153.264
C06942=1094.959,400.534,-96.951,178.679,22.796,153.265
C06943=1094.965,400.780,-96.989,178.682,22.804,153.266
C06944=1094.971,401.027,-97.028,178.684,22.810,153.268
C06945=1094.976,401.275,-97.067,178.688,22.818,153.269
C06946=1094.983,401.521,-97.106,178.690,22.825,153.270
C06947=1094.989,401.768,-97.145,178.692,22.833,153.272
C06948=1094.995,402.015,-97.184,178.696,22.840,153.273
C06949=1095.001,402.262,-97.223,178.698,22.848,153.275
C06950=1095.007,402.509,-97.261,178.701,22.855,153.276
C06951=1095.013,402.756,-97.301,178.704,22.863,153.278
C06952=1095.018,403.002,-97.340,178.707,22.870,153.279
C06953=1095.025,403.249,-97.379,178.709,22.877,153.280
C06954=1095.031,403.496,-97.418,178.713,22.885,153.282
C06955=1095.036,403.743,-97.457,178.715,22.892,153.283
C06956=1095.043,403.990,-97.497,178.718,22.901,153.285
C06957=1095.049,404.237,-97.536,178.720,22.908,153.286
C06958=1095.055,404.483,-97.574,178.724,22.916,153.288
C06959=1095.061,404.730,-97.614,178.726,22.923,153.289
C06960=1095.067,404.977,-97.653,178.729,22.931,153.291
C06961=1095.072,405.224,-97.692,178.731,22.939,153.292
C06962=1095.079,405.471,-97.732,178.735,22.946,153.294
C06963=1095.085,405.718,-97.771,178.737,22.954,153.295
C06964=1095.091,405.965,-97.811,178.740,22.962,153.297
C06965=1095.096,406.211,-97.850,178.743,22.970,153.298
C06966=1095.103,406.458,-97.890,178.745,22.977,153.300
C06967=1095.109,406.705,-97.929,178.749,22.986,153.301
C06968=1095.114,406.952,-97.968,178.751,22.993,153.303
C06969=1095.120,407.198,-98.009,178.754,23.001,153.304
C06970=1095.127,407.445,-98.048,178.756,23.009,153.306
C06971=1095.133,407.693,-98.087,178.759,23.017,153.307
C06972=1095.138,407.939,-98.126,178.762,23.025,153.309
C06973=1095.144,408.186,-98.167,178.764,23.033,153.311
C06974=1095.151,408.433,-98.206,178.768,23.042,153.312
C06975=1095.157,408.679,-98.246,178.771,23.050,153.314
C06976=1095.162,408.926,-98.285,178.773,23.058,153.315
C06977=1095.168,409.173,-98.325,178.776,23.066,153.317
C06978=1095.175,409.419,-98.365,178.779,23.074,153.319
C06979=1095.180,409.667,-98.405,178.781,23.082,153.320
C06980=1095.186,409.913,-98.445,178.784,23.091,153.322
C06981=1095.192,410.160,-98.484,178.787,23.099,153.323
C06982=1095.198,410.380,-98.519,178.790,23.106,153.325
C06983=1095.203,410.600,-98.555,178.792,23.114,153.326
C06984=1095.208,410.820,-98.591,178.794,23.121,153.328
C06985=1095.214,411.040,-98.626,178.797,23.128,153.329
C06986=1095.219,411.260,-98.661,178.799,23.136,153.331
C06987=1095.224,411.480,-98.697,178.801,23.143,153.332
C06988=1095.230,411.699,-98.733,178.804,23.150,153.334
C06989=1095.235,411.919,-98.769,178.806,23.158,153.335
C06990=1095.242,412.167,-98.808,178.809,23.167,153.337
C06991=1095.247,412.413,-98.849,178.812,23.175,153.339
C06992=1095.254,412.660,-98.889,178.815,23.184,153.340
C06993=1095.260,412.907,-98.929,178.818,23.192,153.342
C06994=1095.266,413.154,-98.969,178.820,23.201,153.344
C06995=1095.271,413.400,-99.009,178.823,23.209,153.346
C06996=1095.277,413.646,-99.049,178.826,23.218,153.347
C06997=1095.284,413.893,-99.090,178.829,23.227,153.349
C06998=1095.290,414.139,-99.130,178.832,23.235,153.351
C06999=1095.296,414.387,-99.170,178.834,23.244,153.353
C07000=1095.302,414.633,-99.210,178.837,23.252,153.354
C07001=1095.308,414.880,-99.250,178.840,23.261,153.356
C07002=1095.314,415.126,-99.291,178.843,23.270,153.358
C07003=1095.320,415.373,-99.331,178.846,23.279,153.360
C07004=1095.327,415.619,-99.371,178.848,23.288,153.361
C07005=1095.332,415.866,-99.412,178.851,23.297,153.363
C07006=1095.339,416.113,-99.452,178.853,23.305,153.365
C07007=1095.346,416.360,-99.492,178.856,23.314,153.367
C07008=1095.351,416.607,-99.533,178.859,23.323,153.369
C07009=1095.358,416.853,-99.573,178.862,23.332,153.370
C07010=1095.363,417.100,-99.614,178.865,23.341,153.372
C07011=1095.370,417.347,-99.654,178.867,23.350,153.374
C07012=1095.376,417.593,-99.696,178.870,23.359,153.376
C07013=1095.382,417.839,-99.736,178.873,23.369,153.378
C07014=1095.388,418.086,-99.777,178.876,23.378,153.380
C07015=1095.393,418.333,-99.817,178.878,23.387,153.382
C07016=1095.400,418.580,-99.858,178.881,23.396,153.384
C07017=1095.406,418.826,-99.899,178.884,23.405,153.386
C07018=1095.412,419.072,-99.939,178.887,23.415,153.387
C07019=1095.418,419.319,-99.980,178.890,23.424,153.389
C07020=1095.424,419.565,-100.021,178.892,23.433,153.391
C07021=1095.430,419.812,-100.061,178.895,23.443,153.393
C07022=1095.436,420.059,-100.102,178.898,23.452,153.395
C07023=1095.442,420.305,-100.143,178.901,23.461,153.397
C07024=1095.449,420.552,-100.184,178.903,23.471,153.399
C07025=1095.455,420.798,-100.226,178.906,23.480,153.401
C07026=1095.461,421.045,-100.266,178.909,23.490,153.403
C07027=1095.467,421.291,-100.307,178.911,23.499,153.405
C07028=1095.473,421.538,-100.348,178.914,23.509,153.407
C07029=1095.479,421.784,-100.389,178.917,23.518,153.409
C07030=1095.485,422.031,-100.430,178.919,23.528,153.411
C07031=1095.491,422.277,-100.471,178.922,23.538,153.413
C07032=1095.498,422.523,-100.512,178.925,23.547,153.415
C07033=1095.504,422.770,-100.553,178.928,23.557,153.417
C07034=1095.510,423.016,-100.594,178.931,23.567,153.419
C07035=1095.516,423.264,-100.636,178.934,23.577,153.421
C07036=1095.522,423.510,-100.677,178.936,23.587,153.423
C07037=1095.528,423.756,-100.718,178.939,23.596,153.425
C07038=1095.533,423.984,-100.756,178.942,23.606,153.427
C07039=1095.539,424.210,-100.794,178.943,23.615,153.429
C07040=1095.545,424.438,-100.832,178.946,23.624,153.431
C07041=1095.551,424.665,-100.870,178.949,23.633,153.433
C07042=1095.556,424.892,-100.909,178.952,23.643,153.435
C07043=1095.562,425.119,-100.947,178.954,23.651,153.437
C07044=1095.568,425.346,-100.985,178.957,23.661,153.439
C07045=1095.573,425.573,-101.024,178.959,23.671,153.441
C07046=1095.579,425.819,-101.064,178.962,23.680,153.443
C07047=1095.586,426.066,-101.106,178.964,23.691,153.445
C07048=1095.592,426.312,-101.148,178.967,23.701,153.447
C07049=1095.598,426.558,-101.189,178.970,23.711,153.450
C07050=1095.604,426.805,-101.231,178.973,23.722,153.452
C07051=1095.610,427.052,-101.273,178.975,23.732,153.454
C07052=1095.616,427.298,-101.314,178.978,23.742,153.456
C07053=1095.623,427.545,-101.356,178.981,23.753,153.458
C07054=1095.629,427.791,-101.397,178.983,23.763,153.461
C07055=1095.635,428.037,-101.439,178.986,23.773,153.463
C07056=1095.641,428.284,-101.481,178.988,23.784,153.465
C07057=1095.648,428.530,-101.523,178.992,23.794,153.467
C07058=1095.654,428.777,-101.565,178.994,23.804,153.470
C07059=1095.660,429.023,-101.606,178.997,23.815,153.472
C07060=1095.666,429.269,-101.647,179.000,23.826,153.474
C07061=1095.672,429.516,-101.691,179.002,23.837,153.477
C07062=1095.678,429.762,-101.732,179.005,23.847,153.479
C07063=1095.685,430.009,-101.774,179.008,23.858,153.481
C07064=1095.691,430.254,-101.816,179.010,23.869,153.484
C07065=1095.697,430.500,-101.857,179.014,23.880,153.486
C07066=1095.703,430.747,-101.901,179.016,23.891,153.488
C07067=1095.709,430.993,-101.942,179.018,23.901,153.490
C07068=1095.715,431.240,-101.984,179.021,23.913,153.493
C07069=1095.722,431.486,-102.026,179.024,23.924,153.495
C07070=1095.728,431.733,-102.068,179.027,23.935,153.498
C07071=1095.734,431.978,-102.111,179.029,23.946,153.500
C07072=1095.741,432.225,-102.153,179.032,23.957,153.503
C07073=1095.747,432.471,-102.195,179.035,23.968,153.505
C07074=1095.753,432.717,-102.237,179.037,23.979,153.507
C07075=1095.759,432.964,-102.279,179.040,23.990,153.510
C07076=1095.765,433.210,-102.322,179.043,24.001,153.512
C07077=1095.772,433.456,-102.364,179.046,24.013,153.515
C07078=1095.778,433.702,-102.407,179.048,24.024,153.517
C07079=1095.784,433.948,-102.449,179.051,24.036,153.520
C07080=1095.790,434.195,-102.492,179.053,24.047,153.522
C07081=1095.796,434.441,-102.534,179.056,24.059,153.525
C07082=1095.802,434.687,-102.577,179.059,24.070,153.527
C07083=1095.809,434.933,-102.619,179.062,24.082,153.530
C07084=1095.815,435.179,-102.662,179.064,24.093,153.532
C07085=1095.821,435.426,-102.704,179.067,24.105,153.535
C07086=1095.827,435.672,-102.747,179.069,24.117,153.538
C07087=1095.833,435.918,-102.789,179.072,24.129,153.540
C07088=1095.839,436.164,-102.832,179.075,24.141,153.543
C07089=1095.846,436.411,-102.875,179.077,24.152,153.545
C07090=1095.851,436.657,-102.918,179.080,24.164,153.548
C07091=1095.858,436.903,-102.960,179.082,24.176,153.551
C07092=1095.865,437.149,-103.004,179.086,24.188,153.553
C07093=1095.871,437.394,-103.046,179.088,24.200,153.556
C07094=1095.877,437.648,-103.090,179.090,24.212,153.559
C07095=1095.884,437.901,-103.134,179.093,24.225,153.562
C07096=1095.891,438.154,-103.178,179.096,24.237,153.564
C07097=1095.897,438.407,-103.223,179.099,24.250,153.567
C07098=1095.904,438.653,-103.266,179.101,24.261,153.570
C07099=1095.909,438.899,-103.308,179.104,24.274,153.573
C07100=1095.916,439.145,-103.351,179.107,24.286,153.575
C07101=1095.922,439.391,-103.395,179.110,24.298,153.578
C07102=1095.929,439.639,-103.438,179.112,24.311,153.581
C07103=1095.935,439.886,-103.481,179.115,24.323,153.583
C07104=1095.941,440.134,-103.525,179.118,24.336,153.586
C07105=1095.948,440.381,-103.568,179.121,24.348,153.589
C07106=1095.954,440.627,-103.611,179.123,24.361,153.592
C07107=1095.960,440.873,-103.654,179.125,24.373,153.595
C07108=1095.966,441.119,-103.697,179.128,24.386,153.598
C07109=1095.973,441.365,-103.741,179.131,24.399,153.601
C07110=1095.979,441.612,-103.784,179.133,24.411,153.603
C07111=1095.986,441.857,-103.828,179.136,24.424,153.606
C07112=1095.992,442.103,-103.871,179.139,24.437,153.609
C07113=1095.998,442.349,-103.914,179.142,24.450,153.612
C07114=1096.004,442.595,-103.958,179.143,24.463,153.615
C07115=1096.011,442.841,-104.002,179.146,24.476,153.618
C07116=1096.017,443.087,-104.046,179.149,24.489,153.621
C07117=1096.023,443.334,-104.089,179.152,24.502,153.624
C07118=1096.029,443.579,-104.132,179.154,24.515,153.627
C07119=1096.036,443.825,-104.176,179.157,24.529,153.630
C07120=1096.042,444.071,-104.220,179.159,24.541,153.633
C07121=1096.048,444.317,-104.264,179.162,24.555,153.636
C07122=1096.056,444.563,-104.307,179.163,24.568,153.639
C07123=1096.062,444.809,-104.350,179.166,24.581,153.642
C07124=1096.068,445.055,-104.394,179.168,24.594,153.645
C07125=1096.075,445.301,-104.438,179.170,24.608,153.648
C07126=1096.081,445.547,-104.482,179.170,24.621,153.652
C07127=1096.087,445.793,-104.526,179.172,24.634,153.655
C07128=1096.093,446.039,-104.570,179.173,24.647,153.658
C07129=1096.100,446.285,-104.614,179.174,24.660,153.661
C07130=1096.106,446.531,-104.658,179.175,24.673,153.664
C07131=1096.113,446.777,-104.702,179.175,24.686,153.667
C07132=1096.119,447.023,-104.746,179.176,24.699,153.671
C07133=1096.126,447.269,-104.790,179.177,24.712,153.674
C07134=1096.132,447.515,-104.834,179.177,24.725,153.677
C07135=1096.138,447.761,-104.878,179.177,24.738,153.680
C07136=1096.144,448.007,-104.922,179.177,24.751,153.684
C07137=1096.151,448.253,-104.966,179.177,24.764,153.687
C07138=1096.157,448.498,-105.011,179.177,24.777,153.690
C07139=1096.164,448.744,-105.055,179.177,24.790,153.694
C07140=1096.169,448.990,-105.099,179.175,24.803,153.697
C07141=1096.176,449.236,-105.143,179.175,24.816,153.701
C07142=1096.183,449.482,-105.187,179.174,24.829,153.704
C07143=1096.189,449.728,-105.231,179.174,24.842,153.707
C07144=1096.196,449.973,-105.276,179.173,24.855,153.711
C07145=1096.203,450.219,-105.319,179.172,24.867,153.714
C07146=1095.812,450.212,-105.484,179.116,25.079,153.774
C07147=1095.804,449.965,-105.440,179.117,25.067,153.771
C07148=1095.797,449.719,-105.396,179.118,25.054,153.768
C07149=1095.791,449.474,-105.352,179.118,25.040,153.765
C07150=1095.785,449.228,-105.307,179.119,25.028,153.761
C07151=1095.778,448.982,-105.263,179.119,25.015,153.758
C07152=1095.772,448.736,-105.219,179.120,25.002,153.754
C07153=1095.765,448.490,-105.175,179.120,24.989,153.751
C07154=1095.758,448.244,-105.130,179.120,24.976,153.748
C07155=1095.752,447.998,-105.086,179.120,24.962,153.744
C07156=1095.746,447.752,-105.042,179.120,24.950,153.741
C07157=1095.740,447.506,-104.998,179.120,24.936,153.738
C07158=1095.733,447.261,-104.953,179.120,24.923,153.735
C07159=1095.726,447.015,-104.910,179.119,24.910,153.731
C07160=1095.721,446.768,-104.865,179.119,24.897,153.728
C07161=1095.714,446.522,-104.821,179.118,24.884,153.725
C07162=1095.708,446.276,-104.777,179.117,24.871,153.722
C07163=1095.701,446.031,-104.734,179.115,24.857,153.718
C07164=1095.695,445.785,-104.690,179.115,24.844,153.715
C07165=1095.688,445.539,-104.645,179.113,24.831,153.712
C07166=1095.682,445.293,-104.601,179.112,24.818,153.709
C07167=1095.675,445.047,-104.558,179.110,24.805,153.706
C07168=1095.669,444.801,-104.514,179.108,24.792,153.703
C07169=1095.663,444.555,-104.470,179.105,24.778,153.700
C07170=1095.656,444.309,-104.426,179.103,24.765,153.697
C07171=1095.650,444.063,-104.382,179.101,24.752,153.693
C07172=1095.644,443.817,-104.339,179.099,24.738,153.690
C07173=1095.637,443.571,-104.295,179.096,24.725,153.687
C07174=1095.631,443.325,-104.251,179.093,24.712,153.684
C07175=1095.625,443.080,-104.208,179.090,24.699,153.681
C07176=1095.619,442.834,-104.164,179.087,24.686,153.678
C07177=1095.612,442.588,-104.120,179.086,24.673,153.676
C07178=1095.606,442.341,-104.077,179.083,24.660,153.673
C07179=1095.600,442.095,-104.033,179.080,24.647,153.670
C07180=1095.592,441.849,-103.990,179.077,24.634,153.667
C07181=1095.586,441.603,-103.946,179.074,24.621,153.664
C07182=1095.580,441.357,-103.903,179.072,24.608,153.661
C07183=1095.574,441.112,-103.859,179.069,24.595,153.658
C07184=1095.568,440.865,-103.816,179.066,24.582,153.655
C07185=1095.562,440.619,-103.772,179.063,24.570,153.652
C07186=1095.554,440.373,-103.729,179.061,24.557,153.649
C07187=1095.549,440.127,-103.686,179.058,24.545,153.647
C07188=1095.543,439.881,-103.643,179.055,24.532,153.644
C07189=1095.536,439.635,-103.600,179.052,24.520,153.641
C07190=1095.529,439.389,-103.557,179.050,24.507,153.638
C07191=1095.523,439.144,-103.514,179.047,24.495,153.636
C07192=1095.517,438.898,-103.471,179.044,24.482,153.633
C07193=1095.510,438.652,-103.428,179.042,24.471,153.630
C07194=1095.504,438.407,-103.385,179.039,24.458,153.627
C07195=1095.498,438.162,-103.342,179.037,24.446,153.625
C07196=1095.491,437.917,-103.299,179.034,24.434,153.622
C07197=1095.485,437.671,-103.257,179.031,24.422,153.619
C07198=1095.478,437.426,-103.214,179.028,24.410,153.617
C07199=1095.472,437.180,-103.171,179.025,24.398,153.614
C07200=1095.466,436.934,-103.128,179.023,24.386,153.611
C07201=1095.460,436.688,-103.085,179.020,24.374,153.609
C07202=1095.453,436.443,-103.042,179.017,24.362,153.606
C07203=1095.447,436.196,-102.999,179.015,24.350,153.603
C07204=1095.441,435.949,-102.956,179.012,24.338,153.601
C07205=1095.435,435.704,-102.914,179.010,24.326,153.598
C07206=1095.429,435.457,-102.871,179.006,24.315,153.595
C07207=1095.422,435.211,-102.828,179.004,24.303,153.593
C07208=1095.416,434.965,-102.785,179.001,24.291,153.590
C07209=1095.410,434.719,-102.743,178.999,24.280,153.588
C07210=1095.404,434.472,-102.701,178.996,24.268,153.585
C07211=1095.397,434.226,-102.658,178.992,24.256,153.583
C07212=1095.392,433.980,-102.616,178.990,24.245,153.580
C07213=1095.385,433.734,-102.573,178.987,24.233,153.578
C07214=1095.379,433.488,-102.531,178.985,24.222,153.575
C07215=1095.373,433.242,-102.488,178.982,24.211,153.573
C07216=1095.367,432.995,-102.446,178.979,24.199,153.570
C07217=1095.361,432.749,-102.403,178.977,24.188,153.568
C07218=1095.354,432.503,-102.361,178.974,24.177,153.565
C07219=1095.348,432.256,-102.319,178.971,24.166,153.563
C07220=1095.341,432.010,-102.277,178.968,24.154,153.560
C07221=1095.335,431.764,-102.234,178.966,24.143,153.558
C07222=1095.329,431.517,-102.192,178.962,24.132,153.556
C07223=1095.323,431.272,-102.150,178.960,24.121,153.553
C07224=1095.316,431.025,-102.108,178.958,24.110,153.551
C07225=1095.311,430.779,-102.065,178.954,24.099,153.548
C07226=1095.305,430.533,-102.024,178.952,24.088,153.546
C07227=1095.298,430.286,-101.981,178.949,24.077,153.544
C07228=1095.292,430.040,-101.940,178.946,24.066,153.541
C07229=1095.285,429.794,-101.897,178.944,24.056,153.539
C07230=1095.280,429.547,-101.855,178.940,24.045,153.537
C07231=1095.273,429.301,-101.813,178.938,24.034,153.534
C07232=1095.267,429.055,-101.771,178.935,24.023,153.532
C07233=1095.261,428.809,-101.730,178.933,24.013,153.530
C07234=1095.254,428.562,-101.688,178.929,24.002,153.527
C07235=1095.248,428.316,-101.646,178.927,23.992,153.525
C07236=1095.242,428.069,-101.604,178.924,23.981,153.523
C07237=1095.236,427.823,-101.562,178.921,23.970,153.521
C07238=1095.229,427.576,-101.521,178.919,23.960,153.518
C07239=1095.223,427.330,-101.479,178.916,23.950,153.516
C07240=1095.217,427.084,-101.438,178.913,23.939,153.514
C07241=1095.210,426.838,-101.395,178.910,23.929,153.512
C07242=1095.204,426.591,-101.354,178.907,23.919,153.510
C07243=1095.199,426.345,-101.312,178.905,23.908,153.507
C07244=1095.192,426.098,-101.270,178.902,23.898,153.505
C07245=1095.186,425.852,-101.229,178.899,23.888,153.503
C07246=1095.180,425.606,-101.187,178.896,23.877,153.501
C07247=1095.174,425.378,-101.149,178.893,23.868,153.499
C07248=1095.169,425.151,-101.111,178.891,23.859,153.497
C07249=1095.162,424.923,-101.073,178.889,23.849,153.495
C07250=1095.157,424.695,-101.034,178.886,23.840,153.493
C07251=1095.152,424.468,-100.996,178.884,23.831,153.491
C07252=1095.146,424.240,-100.957,178.881,23.821,153.489
C07253=1095.140,424.013,-100.920,178.878,23.812,153.487
C07254=1095.135,423.785,-100.882,178.876,23.803,153.485
C07255=1095.128,423.538,-100.840,178.873,23.793,153.483
C07256=1095.122,423.292,-100.799,178.870,23.783,153.481
C07257=1095.116,423.046,-100.757,178.867,23.773,153.479
C07258=1095.111,422.799,-100.717,178.865,23.763,153.477
C07259=1095.104,422.552,-100.675,178.862,23.753,153.475
C07260=1095.097,422.306,-100.634,178.859,23.744,153.473
C07261=1095.092,422.059,-100.593,178.857,23.734,153.471
C07262=1095.086,421.813,-100.552,178.854,23.725,153.469
C07263=1095.079,421.567,-100.510,178.851,23.715,153.467
C07264=1095.073,421.320,-100.470,178.847,23.705,153.465
C07265=1095.067,421.074,-100.428,178.845,23.696,153.463
C07266=1095.061,420.827,-100.388,178.842,23.686,153.461
C07267=1095.055,420.581,-100.347,178.839,23.676,153.459
C07268=1095.049,420.334,-100.306,178.836,23.667,153.457
C07269=1095.042,420.087,-100.265,178.834,23.657,153.455
C07270=1095.036,419.841,-100.224,178.831,23.648,153.453
C07271=1095.030,419.594,-100.183,178.828,23.639,153.451
